RoboDK station: plane_optimization.rdk

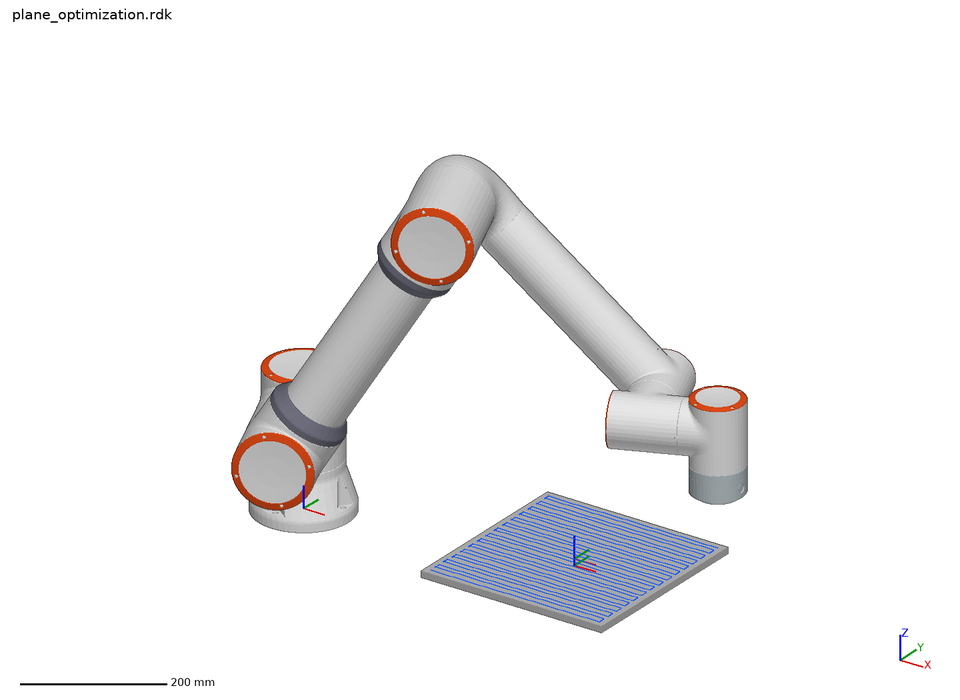
[picture v0: the station drawn from its stored meshes, robots at their saved joint values, targets as dots, program paths as lines]
Station plane_optimization (saved by RoboDK 6.0.4). Poses are relative to the parent item; angles as X-Y-Z fixed-axis rotations.
  - frame FAIRINO FR5 Base at (0, 0, 0) mm
    - robot FAIRINO FR5: 6 axes
        modified DH rows (alpha deg, a mm, theta deg, d mm): 0, 0, 0, 152; 90, 0, 180, 0; 0, 425, 0, 0; 0, 395, 0, 102; -90, 0, 0, 102; 90, 0, 180, 100
        joint limits [-175, -265, -160, -265, -175, -175] to [175, 85, 160, 85, 175, 175]; home [0, -90, -90, 0, 90, 0]; saved at [23.033, -121.455, -104.631, -43.915, 90, 23.033]
      - tool Tool 1, TCP at (0, 0, 80) mm
  - frame PlateFrame at (450, 0, 50) mm
    - target Home (Cartesian target) at (45, -102, 629) mm, rotated rx -90 ry 0 rz -90 deg; joints [0, -90, -90, 0, 90, 0] of FAIRINO FR5
    - target Target_001 (Cartesian target) at (-140, -140, 0) mm, rotated rx -180 ry 0 rz -90 deg; joints [-6.855, -94.267, -146.837, -28.896, 90, -6.855] of FAIRINO FR5
    - target Target_002 (Cartesian target) at (-130, -140, 0) mm, rotated rx -180 ry 0 rz -90 deg; joints [-6.65, -95.39, -145.504, -29.106, 90, -6.65] of FAIRINO FR5
    - target Target_003 (Cartesian target) at (-120, -140, 0) mm, rotated rx -180 ry 0 rz -90 deg; joints [-6.457, -96.486, -144.158, -29.356, 90, -6.457] of FAIRINO FR5
    - target Target_004 (Cartesian target) at (-110, -140, 0) mm, rotated rx -180 ry 0 rz -90 deg; joints [-6.275, -97.559, -142.799, -29.642, 90, -6.275] of FAIRINO FR5
    - target Target_005 (Cartesian target) at (-100, -140, 0) mm, rotated rx -180 ry 0 rz -90 deg; joints [-6.102, -98.61, -141.428, -29.962, 90, -6.102] of FAIRINO FR5
    - target Target_006 (Cartesian target) at (-90, -140, 0) mm, rotated rx -180 ry 0 rz -90 deg; joints [-5.939, -99.642, -140.044, -30.313, 90, -5.939] of FAIRINO FR5
    - target Target_007 (Cartesian target) at (-80, -140, 0) mm, rotated rx -180 ry 0 rz -90 deg; joints [-5.784, -100.658, -138.649, -30.693, 90, -5.784] of FAIRINO FR5
    - target Target_008 (Cartesian target) at (-70, -140, 0) mm, rotated rx -180 ry 0 rz -90 deg; joints [-5.637, -101.66, -137.242, -31.099, 90, -5.637] of FAIRINO FR5
    - target Target_009 (Cartesian target) at (-60, -140, 0) mm, rotated rx -180 ry 0 rz -90 deg; joints [-5.497, -102.648, -135.823, -31.529, 90, -5.497] of FAIRINO FR5
    - target Target_010 (Cartesian target) at (-50, -140, 0) mm, rotated rx -180 ry 0 rz -90 deg; joints [-5.363, -103.625, -134.392, -31.983, 90, -5.363] of FAIRINO FR5
    - target Target_011 (Cartesian target) at (-40, -140, 0) mm, rotated rx -180 ry 0 rz -90 deg; joints [-5.236, -104.592, -132.949, -32.459, 90, -5.236] of FAIRINO FR5
    - target Target_012 (Cartesian target) at (-30, -140, 0) mm, rotated rx -180 ry 0 rz -90 deg; joints [-5.115, -105.55, -131.495, -32.955, 90, -5.115] of FAIRINO FR5
    - target Target_013 (Cartesian target) at (-20, -140, 0) mm, rotated rx -180 ry 0 rz -90 deg; joints [-4.999, -106.501, -130.028, -33.471, 90, -4.999] of FAIRINO FR5
    - target Target_014 (Cartesian target) at (-10, -140, 0) mm, rotated rx -180 ry 0 rz -90 deg; joints [-4.888, -107.446, -128.549, -34.005, 90, -4.888] of FAIRINO FR5
    - target Target_015 (Cartesian target) at (0, -140, 0) mm, rotated rx -180 ry 0 rz -90 deg; joints [-4.782, -108.386, -127.057, -34.557, 90, -4.782] of FAIRINO FR5
    - target Target_016 (Cartesian target) at (10, -140, 0) mm, rotated rx -180 ry 0 rz -90 deg; joints [-4.68, -109.321, -125.553, -35.126, 90, -4.68] of FAIRINO FR5
    - target Target_017 (Cartesian target) at (20, -140, 0) mm, rotated rx -180 ry 0 rz -90 deg; joints [-4.583, -110.253, -124.035, -35.712, 90, -4.583] of FAIRINO FR5
    - target Target_018 (Cartesian target) at (30, -140, 0) mm, rotated rx -180 ry 0 rz -90 deg; joints [-4.489, -111.182, -122.505, -36.314, 90, -4.489] of FAIRINO FR5
    - target Target_019 (Cartesian target) at (40, -140, 0) mm, rotated rx -180 ry 0 rz -90 deg; joints [-4.399, -112.109, -120.96, -36.931, 90, -4.399] of FAIRINO FR5
    - target Target_020 (Cartesian target) at (50, -140, 0) mm, rotated rx -180 ry 0 rz -90 deg; joints [-4.313, -113.036, -119.401, -37.563, 90, -4.313] of FAIRINO FR5
    - target Target_021 (Cartesian target) at (60, -140, 0) mm, rotated rx -180 ry 0 rz -90 deg; joints [-4.23, -113.963, -117.827, -38.21, 90, -4.23] of FAIRINO FR5
    - target Target_022 (Cartesian target) at (70, -140, 0) mm, rotated rx -180 ry 0 rz -90 deg; joints [-4.15, -114.89, -116.238, -38.872, 90, -4.15] of FAIRINO FR5
    - target Target_023 (Cartesian target) at (80, -140, 0) mm, rotated rx -180 ry 0 rz -90 deg; joints [-4.073, -115.818, -114.633, -39.549, 90, -4.073] of FAIRINO FR5
    - target Target_024 (Cartesian target) at (90, -140, 0) mm, rotated rx -180 ry 0 rz -90 deg; joints [-3.999, -116.749, -113.011, -40.24, 90, -3.999] of FAIRINO FR5
    - target Target_025 (Cartesian target) at (100, -140, 0) mm, rotated rx -180 ry 0 rz -90 deg; joints [-3.927, -117.682, -111.373, -40.946, 90, -3.927] of FAIRINO FR5
    - target Target_026 (Cartesian target) at (110, -140, 0) mm, rotated rx -180 ry 0 rz -90 deg; joints [-3.858, -118.618, -109.716, -41.666, 90, -3.858] of FAIRINO FR5
    - target Target_027 (Cartesian target) at (120, -140, 0) mm, rotated rx -180 ry 0 rz -90 deg; joints [-3.792, -119.559, -108.041, -42.401, 90, -3.792] of FAIRINO FR5
    - target Target_028 (Cartesian target) at (130, -140, 0) mm, rotated rx -180 ry 0 rz -90 deg; joints [-3.727, -120.504, -106.346, -43.15, 90, -3.727] of FAIRINO FR5
    - target Target_029 (Cartesian target) at (140, -140, 0) mm, rotated rx -180 ry 0 rz -90 deg; joints [-3.665, -121.455, -104.631, -43.915, 90, -3.665] of FAIRINO FR5
    - target Target_030 (Cartesian target) at (140, -130, 0) mm, rotated rx -180 ry 0 rz -90 deg; joints [-2.706, -121.236, -105.026, -43.738, 90, -2.706] of FAIRINO FR5
    - target Target_031 (Cartesian target) at (130, -130, 0) mm, rotated rx -180 ry 0 rz -90 deg; joints [-2.752, -120.283, -106.743, -42.974, 90, -2.752] of FAIRINO FR5
    - target Target_032 (Cartesian target) at (120, -130, 0) mm, rotated rx -180 ry 0 rz -90 deg; joints [-2.8, -119.335, -108.44, -42.225, 90, -2.8] of FAIRINO FR5
    - target Target_033 (Cartesian target) at (110, -130, 0) mm, rotated rx -180 ry 0 rz -90 deg; joints [-2.85, -118.391, -110.118, -41.491, 90, -2.85] of FAIRINO FR5
    - target Target_034 (Cartesian target) at (100, -130, 0) mm, rotated rx -180 ry 0 rz -90 deg; joints [-2.901, -117.452, -111.777, -40.771, 90, -2.901] of FAIRINO FR5
    - target Target_035 (Cartesian target) at (90, -130, 0) mm, rotated rx -180 ry 0 rz -90 deg; joints [-2.954, -116.515, -113.419, -40.066, 90, -2.954] of FAIRINO FR5
    - target Target_036 (Cartesian target) at (80, -130, 0) mm, rotated rx -180 ry 0 rz -90 deg; joints [-3.009, -115.581, -115.044, -39.375, 90, -3.009] of FAIRINO FR5
    - target Target_037 (Cartesian target) at (70, -130, 0) mm, rotated rx -180 ry 0 rz -90 deg; joints [-3.066, -114.648, -116.653, -38.699, 90, -3.066] of FAIRINO FR5
    - target Target_038 (Cartesian target) at (60, -130, 0) mm, rotated rx -180 ry 0 rz -90 deg; joints [-3.125, -113.717, -118.246, -38.037, 90, -3.125] of FAIRINO FR5
    - target Target_039 (Cartesian target) at (50, -130, 0) mm, rotated rx -180 ry 0 rz -90 deg; joints [-3.187, -112.785, -119.824, -37.39, 90, -3.187] of FAIRINO FR5
    - target Target_040 (Cartesian target) at (40, -130, 0) mm, rotated rx -180 ry 0 rz -90 deg; joints [-3.251, -111.853, -121.388, -36.759, 90, -3.251] of FAIRINO FR5
    - target Target_041 (Cartesian target) at (30, -130, 0) mm, rotated rx -180 ry 0 rz -90 deg; joints [-3.318, -110.92, -122.938, -36.142, 90, -3.318] of FAIRINO FR5
    - target Target_042 (Cartesian target) at (20, -130, 0) mm, rotated rx -180 ry 0 rz -90 deg; joints [-3.388, -109.984, -124.474, -35.542, 90, -3.388] of FAIRINO FR5
    - target Target_043 (Cartesian target) at (10, -130, 0) mm, rotated rx -180 ry 0 rz -90 deg; joints [-3.46, -109.046, -125.997, -34.957, 90, -3.46] of FAIRINO FR5
    - target Target_044 (Cartesian target) at (0, -130, 0) mm, rotated rx -180 ry 0 rz -90 deg; joints [-3.536, -108.103, -127.508, -34.389, 90, -3.536] of FAIRINO FR5
    - target Target_045 (Cartesian target) at (-10, -130, 0) mm, rotated rx -180 ry 0 rz -90 deg; joints [-3.615, -107.156, -129.006, -33.839, 90, -3.615] of FAIRINO FR5
    - target Target_046 (Cartesian target) at (-20, -130, 0) mm, rotated rx -180 ry 0 rz -90 deg; joints [-3.697, -106.202, -130.491, -33.306, 90, -3.697] of FAIRINO FR5
    - target Target_047 (Cartesian target) at (-30, -130, 0) mm, rotated rx -180 ry 0 rz -90 deg; joints [-3.784, -105.242, -131.965, -32.793, 90, -3.784] of FAIRINO FR5
    - target Target_048 (Cartesian target) at (-40, -130, 0) mm, rotated rx -180 ry 0 rz -90 deg; joints [-3.874, -104.273, -133.428, -32.299, 90, -3.874] of FAIRINO FR5
    - target Target_049 (Cartesian target) at (-50, -130, 0) mm, rotated rx -180 ry 0 rz -90 deg; joints [-3.969, -103.295, -134.878, -31.827, 90, -3.969] of FAIRINO FR5
    - target Target_050 (Cartesian target) at (-60, -130, 0) mm, rotated rx -180 ry 0 rz -90 deg; joints [-4.069, -102.306, -136.318, -31.377, 90, -4.069] of FAIRINO FR5
    - target Target_051 (Cartesian target) at (-70, -130, 0) mm, rotated rx -180 ry 0 rz -90 deg; joints [-4.174, -101.304, -137.745, -30.951, 90, -4.174] of FAIRINO FR5
    - target Target_052 (Cartesian target) at (-80, -130, 0) mm, rotated rx -180 ry 0 rz -90 deg; joints [-4.284, -100.288, -139.162, -30.55, 90, -4.284] of FAIRINO FR5
    - target Target_053 (Cartesian target) at (-90, -130, 0) mm, rotated rx -180 ry 0 rz -90 deg; joints [-4.4, -99.255, -140.567, -30.177, 90, -4.4] of FAIRINO FR5
    - target Target_054 (Cartesian target) at (-100, -130, 0) mm, rotated rx -180 ry 0 rz -90 deg; joints [-4.522, -98.205, -141.961, -29.834, 90, -4.522] of FAIRINO FR5
    - target Target_055 (Cartesian target) at (-110, -130, 0) mm, rotated rx -180 ry 0 rz -90 deg; joints [-4.651, -97.133, -143.343, -29.524, 90, -4.651] of FAIRINO FR5
    - target Target_056 (Cartesian target) at (-120, -130, 0) mm, rotated rx -180 ry 0 rz -90 deg; joints [-4.788, -96.038, -144.714, -29.248, 90, -4.788] of FAIRINO FR5
    - target Target_057 (Cartesian target) at (-130, -130, 0) mm, rotated rx -180 ry 0 rz -90 deg; joints [-4.933, -94.917, -146.072, -29.012, 90, -4.933] of FAIRINO FR5
    - target Target_058 (Cartesian target) at (-140, -130, 0) mm, rotated rx -180 ry 0 rz -90 deg; joints [-5.087, -93.765, -147.417, -28.818, 90, -5.087] of FAIRINO FR5
    - target Target_059 (Cartesian target) at (-140, -120, 0) mm, rotated rx -180 ry 0 rz -90 deg; joints [-3.292, -93.288, -147.96, -28.752, 90, -3.292] of FAIRINO FR5
    - target Target_060 (Cartesian target) at (-130, -120, 0) mm, rotated rx -180 ry 0 rz -90 deg; joints [-3.191, -94.468, -146.602, -28.93, 90, -3.191] of FAIRINO FR5
    - target Target_061 (Cartesian target) at (-120, -120, 0) mm, rotated rx -180 ry 0 rz -90 deg; joints [-3.096, -95.614, -145.233, -29.153, 90, -3.096] of FAIRINO FR5
    - target Target_062 (Cartesian target) at (-110, -120, 0) mm, rotated rx -180 ry 0 rz -90 deg; joints [-3.007, -96.731, -143.851, -29.417, 90, -3.007] of FAIRINO FR5
    - target Target_063 (Cartesian target) at (-100, -120, 0) mm, rotated rx -180 ry 0 rz -90 deg; joints [-2.922, -97.822, -142.459, -29.719, 90, -2.922] of FAIRINO FR5
    - target Target_064 (Cartesian target) at (-90, -120, 0) mm, rotated rx -180 ry 0 rz -90 deg; joints [-2.842, -98.891, -141.055, -30.054, 90, -2.842] of FAIRINO FR5
    - target Target_065 (Cartesian target) at (-80, -120, 0) mm, rotated rx -180 ry 0 rz -90 deg; joints [-2.767, -99.939, -139.64, -30.42, 90, -2.767] of FAIRINO FR5
    - target Target_066 (Cartesian target) at (-70, -120, 0) mm, rotated rx -180 ry 0 rz -90 deg; joints [-2.695, -100.97, -138.215, -30.816, 90, -2.695] of FAIRINO FR5
    - target Target_067 (Cartesian target) at (-60, -120, 0) mm, rotated rx -180 ry 0 rz -90 deg; joints [-2.627, -101.985, -136.778, -31.237, 90, -2.627] of FAIRINO FR5
    - target Target_068 (Cartesian target) at (-50, -120, 0) mm, rotated rx -180 ry 0 rz -90 deg; joints [-2.562, -102.986, -135.331, -31.683, 90, -2.562] of FAIRINO FR5
    - target Target_069 (Cartesian target) at (-40, -120, 0) mm, rotated rx -180 ry 0 rz -90 deg; joints [-2.5, -103.975, -133.873, -32.152, 90, -2.5] of FAIRINO FR5
    - target Target_070 (Cartesian target) at (-30, -120, 0) mm, rotated rx -180 ry 0 rz -90 deg; joints [-2.441, -104.953, -132.403, -32.643, 90, -2.441] of FAIRINO FR5
    - target Target_071 (Cartesian target) at (-20, -120, 0) mm, rotated rx -180 ry 0 rz -90 deg; joints [-2.385, -105.923, -130.922, -33.155, 90, -2.385] of FAIRINO FR5
    - target Target_072 (Cartesian target) at (-10, -120, 0) mm, rotated rx -180 ry 0 rz -90 deg; joints [-2.332, -106.885, -129.43, -33.685, 90, -2.332] of FAIRINO FR5
    - target Target_073 (Cartesian target) at (0, -120, 0) mm, rotated rx -180 ry 0 rz -90 deg; joints [-2.28, -107.84, -127.926, -34.234, 90, -2.28] of FAIRINO FR5
    - target Target_074 (Cartesian target) at (10, -120, 0) mm, rotated rx -180 ry 0 rz -90 deg; joints [-2.231, -108.789, -126.41, -34.801, 90, -2.231] of FAIRINO FR5
    - target Target_075 (Cartesian target) at (20, -120, 0) mm, rotated rx -180 ry 0 rz -90 deg; joints [-2.184, -109.734, -124.882, -35.384, 90, -2.184] of FAIRINO FR5
    - target Target_076 (Cartesian target) at (30, -120, 0) mm, rotated rx -180 ry 0 rz -90 deg; joints [-2.139, -110.676, -123.34, -35.984, 90, -2.139] of FAIRINO FR5
    - target Target_077 (Cartesian target) at (40, -120, 0) mm, rotated rx -180 ry 0 rz -90 deg; joints [-2.096, -111.615, -121.786, -36.6, 90, -2.096] of FAIRINO FR5
    - target Target_078 (Cartesian target) at (50, -120, 0) mm, rotated rx -180 ry 0 rz -90 deg; joints [-2.054, -112.552, -120.218, -37.231, 90, -2.054] of FAIRINO FR5
    - target Target_079 (Cartesian target) at (60, -120, 0) mm, rotated rx -180 ry 0 rz -90 deg; joints [-2.014, -113.488, -118.635, -37.877, 90, -2.014] of FAIRINO FR5
    - target Target_080 (Cartesian target) at (70, -120, 0) mm, rotated rx -180 ry 0 rz -90 deg; joints [-1.976, -114.424, -117.038, -38.538, 90, -1.976] of FAIRINO FR5
    - target Target_081 (Cartesian target) at (80, -120, 0) mm, rotated rx -180 ry 0 rz -90 deg; joints [-1.939, -115.36, -115.426, -39.214, 90, -1.939] of FAIRINO FR5
    - target Target_082 (Cartesian target) at (90, -120, 0) mm, rotated rx -180 ry 0 rz -90 deg; joints [-1.903, -116.298, -113.798, -39.904, 90, -1.903] of FAIRINO FR5
    - target Target_083 (Cartesian target) at (100, -120, 0) mm, rotated rx -180 ry 0 rz -90 deg; joints [-1.869, -117.238, -112.153, -40.609, 90, -1.869] of FAIRINO FR5
    - target Target_084 (Cartesian target) at (110, -120, 0) mm, rotated rx -180 ry 0 rz -90 deg; joints [-1.836, -118.181, -110.491, -41.328, 90, -1.836] of FAIRINO FR5
    - target Target_085 (Cartesian target) at (120, -120, 0) mm, rotated rx -180 ry 0 rz -90 deg; joints [-1.804, -119.127, -108.81, -42.062, 90, -1.804] of FAIRINO FR5
    - target Target_086 (Cartesian target) at (130, -120, 0) mm, rotated rx -180 ry 0 rz -90 deg; joints [-1.773, -120.078, -107.111, -42.811, 90, -1.773] of FAIRINO FR5
    - target Target_087 (Cartesian target) at (140, -120, 0) mm, rotated rx -180 ry 0 rz -90 deg; joints [-1.743, -121.033, -105.392, -43.575, 90, -1.743] of FAIRINO FR5
    - target Target_088 (Cartesian target) at (140, -110, 0) mm, rotated rx -180 ry 0 rz -90 deg; joints [-0.776, -120.846, -105.729, -43.424, 90, -0.776] of FAIRINO FR5
    - target Target_089 (Cartesian target) at (130, -110, 0) mm, rotated rx -180 ry 0 rz -90 deg; joints [-0.789, -119.889, -107.45, -42.661, 90, -0.789] of FAIRINO FR5
    - target Target_090 (Cartesian target) at (120, -110, 0) mm, rotated rx -180 ry 0 rz -90 deg; joints [-0.803, -118.936, -109.152, -41.913, 90, -0.803] of FAIRINO FR5
    - target Target_091 (Cartesian target) at (110, -110, 0) mm, rotated rx -180 ry 0 rz -90 deg; joints [-0.817, -117.987, -110.834, -41.179, 90, -0.817] of FAIRINO FR5
    - target Target_092 (Cartesian target) at (100, -110, 0) mm, rotated rx -180 ry 0 rz -90 deg; joints [-0.832, -117.041, -112.499, -40.46, 90, -0.832] of FAIRINO FR5
    - target Target_093 (Cartesian target) at (90, -110, 0) mm, rotated rx -180 ry 0 rz -90 deg; joints [-0.848, -116.098, -114.147, -39.755, 90, -0.848] of FAIRINO FR5
    - target Target_094 (Cartesian target) at (80, -110, 0) mm, rotated rx -180 ry 0 rz -90 deg; joints [-0.864, -115.157, -115.778, -39.066, 90, -0.864] of FAIRINO FR5
    - target Target_095 (Cartesian target) at (70, -110, 0) mm, rotated rx -180 ry 0 rz -90 deg; joints [-0.88, -114.216, -117.393, -38.39, 90, -0.88] of FAIRINO FR5
    - target Target_096 (Cartesian target) at (60, -110, 0) mm, rotated rx -180 ry 0 rz -90 deg; joints [-0.897, -113.276, -118.994, -37.729, 90, -0.897] of FAIRINO FR5
    - target Target_097 (Cartesian target) at (50, -110, 0) mm, rotated rx -180 ry 0 rz -90 deg; joints [-0.915, -112.336, -120.58, -37.084, 90, -0.915] of FAIRINO FR5
    - target Target_098 (Cartesian target) at (40, -110, 0) mm, rotated rx -180 ry 0 rz -90 deg; joints [-0.934, -111.394, -122.153, -36.453, 90, -0.934] of FAIRINO FR5
    - target Target_099 (Cartesian target) at (30, -110, 0) mm, rotated rx -180 ry 0 rz -90 deg; joints [-0.953, -110.45, -123.712, -35.838, 90, -0.953] of FAIRINO FR5
    - target Target_100 (Cartesian target) at (20, -110, 0) mm, rotated rx -180 ry 0 rz -90 deg; joints [-0.973, -109.503, -125.258, -35.239, 90, -0.973] of FAIRINO FR5
    - target Target_101 (Cartesian target) at (10, -110, 0) mm, rotated rx -180 ry 0 rz -90 deg; joints [-0.994, -108.552, -126.791, -34.657, 90, -0.994] of FAIRINO FR5
    - target Target_102 (Cartesian target) at (0, -110, 0) mm, rotated rx -180 ry 0 rz -90 deg; joints [-1.016, -107.596, -128.313, -34.092, 90, -1.016] of FAIRINO FR5
    - target Target_103 (Cartesian target) at (-10, -110, 0) mm, rotated rx -180 ry 0 rz -90 deg; joints [-1.039, -106.633, -129.823, -33.544, 90, -1.039] of FAIRINO FR5
    - target Target_104 (Cartesian target) at (-20, -110, 0) mm, rotated rx -180 ry 0 rz -90 deg; joints [-1.064, -105.664, -131.321, -33.015, 90, -1.064] of FAIRINO FR5
    - target Target_105 (Cartesian target) at (-30, -110, 0) mm, rotated rx -180 ry 0 rz -90 deg; joints [-1.089, -104.686, -132.808, -32.506, 90, -1.089] of FAIRINO FR5
    - target Target_106 (Cartesian target) at (-40, -110, 0) mm, rotated rx -180 ry 0 rz -90 deg; joints [-1.115, -103.698, -134.284, -32.018, 90, -1.115] of FAIRINO FR5
    - target Target_107 (Cartesian target) at (-50, -110, 0) mm, rotated rx -180 ry 0 rz -90 deg; joints [-1.143, -102.698, -135.75, -31.552, 90, -1.143] of FAIRINO FR5
    - target Target_108 (Cartesian target) at (-60, -110, 0) mm, rotated rx -180 ry 0 rz -90 deg; joints [-1.172, -101.686, -137.205, -31.11, 90, -1.172] of FAIRINO FR5
    - target Target_109 (Cartesian target) at (-70, -110, 0) mm, rotated rx -180 ry 0 rz -90 deg; joints [-1.203, -100.658, -138.649, -30.693, 90, -1.203] of FAIRINO FR5
    - target Target_110 (Cartesian target) at (-80, -110, 0) mm, rotated rx -180 ry 0 rz -90 deg; joints [-1.235, -99.614, -140.083, -30.303, 90, -1.235] of FAIRINO FR5
    - target Target_111 (Cartesian target) at (-90, -110, 0) mm, rotated rx -180 ry 0 rz -90 deg; joints [-1.269, -98.55, -141.507, -29.943, 90, -1.269] of FAIRINO FR5
    - target Target_112 (Cartesian target) at (-100, -110, 0) mm, rotated rx -180 ry 0 rz -90 deg; joints [-1.305, -97.465, -142.92, -29.615, 90, -1.305] of FAIRINO FR5
    - target Target_113 (Cartesian target) at (-110, -110, 0) mm, rotated rx -180 ry 0 rz -90 deg; joints [-1.343, -96.355, -144.322, -29.323, 90, -1.343] of FAIRINO FR5
    - target Target_114 (Cartesian target) at (-120, -110, 0) mm, rotated rx -180 ry 0 rz -90 deg; joints [-1.384, -95.216, -145.714, -29.07, 90, -1.384] of FAIRINO FR5
    - target Target_115 (Cartesian target) at (-130, -110, 0) mm, rotated rx -180 ry 0 rz -90 deg; joints [-1.426, -94.045, -147.094, -28.86, 90, -1.426] of FAIRINO FR5
    - target Target_116 (Cartesian target) at (-140, -110, 0) mm, rotated rx -180 ry 0 rz -90 deg; joints [-1.472, -92.838, -148.463, -28.698, 90, -1.472] of FAIRINO FR5
    - target Target_117 (Cartesian target) at (-140, -100, 0) mm, rotated rx -180 ry 0 rz -90 deg; joints [0.37, -92.418, -148.927, -28.655, 90, 0.37] of FAIRINO FR5
    - target Target_118 (Cartesian target) at (-130, -100, 0) mm, rotated rx -180 ry 0 rz -90 deg; joints [0.358, -93.652, -147.547, -28.801, 90, 0.358] of FAIRINO FR5
    - target Target_119 (Cartesian target) at (-120, -100, 0) mm, rotated rx -180 ry 0 rz -90 deg; joints [0.348, -94.845, -146.156, -28.998, 90, 0.348] of FAIRINO FR5
    - target Target_120 (Cartesian target) at (-110, -100, 0) mm, rotated rx -180 ry 0 rz -90 deg; joints [0.337, -96.005, -144.755, -29.24, 90, 0.337] of FAIRINO FR5
    - target Target_121 (Cartesian target) at (-100, -100, 0) mm, rotated rx -180 ry 0 rz -90 deg; joints [0.328, -97.133, -143.343, -29.524, 90, 0.328] of FAIRINO FR5
    - target Target_122 (Cartesian target) at (-90, -100, 0) mm, rotated rx -180 ry 0 rz -90 deg; joints [0.319, -98.235, -141.922, -29.844, 90, 0.319] of FAIRINO FR5
    - target Target_123 (Cartesian target) at (-80, -100, 0) mm, rotated rx -180 ry 0 rz -90 deg; joints [0.31, -99.313, -140.49, -30.197, 90, 0.31] of FAIRINO FR5
    - target Target_124 (Cartesian target) at (-70, -100, 0) mm, rotated rx -180 ry 0 rz -90 deg; joints [0.302, -100.37, -139.048, -30.582, 90, 0.302] of FAIRINO FR5
    - target Target_125 (Cartesian target) at (-60, -100, 0) mm, rotated rx -180 ry 0 rz -90 deg; joints [0.294, -101.41, -137.596, -30.994, 90, 0.294] of FAIRINO FR5
    - target Target_126 (Cartesian target) at (-50, -100, 0) mm, rotated rx -180 ry 0 rz -90 deg; joints [0.287, -102.433, -136.134, -31.433, 90, 0.287] of FAIRINO FR5
    - target Target_127 (Cartesian target) at (-40, -100, 0) mm, rotated rx -180 ry 0 rz -90 deg; joints [0.28, -103.442, -134.662, -31.896, 90, 0.28] of FAIRINO FR5
    - target Target_128 (Cartesian target) at (-30, -100, 0) mm, rotated rx -180 ry 0 rz -90 deg; joints [0.273, -104.439, -133.179, -32.382, 90, 0.273] of FAIRINO FR5
    - target Target_129 (Cartesian target) at (-20, -100, 0) mm, rotated rx -180 ry 0 rz -90 deg; joints [0.267, -105.425, -131.686, -32.889, 90, 0.267] of FAIRINO FR5
    - target Target_130 (Cartesian target) at (-10, -100, 0) mm, rotated rx -180 ry 0 rz -90 deg; joints [0.261, -106.402, -130.182, -33.416, 90, 0.261] of FAIRINO FR5
    - target Target_131 (Cartesian target) at (0, -100, 0) mm, rotated rx -180 ry 0 rz -90 deg; joints [0.255, -107.371, -128.667, -33.962, 90, 0.255] of FAIRINO FR5
    - target Target_132 (Cartesian target) at (10, -100, 0) mm, rotated rx -180 ry 0 rz -90 deg; joints [0.249, -108.333, -127.141, -34.526, 90, 0.249] of FAIRINO FR5
    - target Target_133 (Cartesian target) at (20, -100, 0) mm, rotated rx -180 ry 0 rz -90 deg; joints [0.244, -109.29, -125.602, -35.108, 90, 0.244] of FAIRINO FR5
    - target Target_134 (Cartesian target) at (30, -100, 0) mm, rotated rx -180 ry 0 rz -90 deg; joints [0.239, -110.243, -124.052, -35.706, 90, 0.239] of FAIRINO FR5
    - target Target_135 (Cartesian target) at (40, -100, 0) mm, rotated rx -180 ry 0 rz -90 deg; joints [0.234, -111.192, -122.489, -36.32, 90, 0.234] of FAIRINO FR5
    - target Target_136 (Cartesian target) at (50, -100, 0) mm, rotated rx -180 ry 0 rz -90 deg; joints [0.229, -112.138, -120.912, -36.95, 90, 0.229] of FAIRINO FR5
    - target Target_137 (Cartesian target) at (60, -100, 0) mm, rotated rx -180 ry 0 rz -90 deg; joints [0.225, -113.082, -119.323, -37.595, 90, 0.225] of FAIRINO FR5
    - target Target_138 (Cartesian target) at (70, -100, 0) mm, rotated rx -180 ry 0 rz -90 deg; joints [0.22, -114.026, -117.719, -38.255, 90, 0.22] of FAIRINO FR5
    - target Target_139 (Cartesian target) at (80, -100, 0) mm, rotated rx -180 ry 0 rz -90 deg; joints [0.216, -114.97, -116.1, -38.93, 90, 0.216] of FAIRINO FR5
    - target Target_140 (Cartesian target) at (90, -100, 0) mm, rotated rx -180 ry 0 rz -90 deg; joints [0.212, -115.914, -114.466, -39.62, 90, 0.212] of FAIRINO FR5
    - target Target_141 (Cartesian target) at (100, -100, 0) mm, rotated rx -180 ry 0 rz -90 deg; joints [0.208, -116.861, -112.815, -40.324, 90, 0.208] of FAIRINO FR5
    - target Target_142 (Cartesian target) at (110, -100, 0) mm, rotated rx -180 ry 0 rz -90 deg; joints [0.205, -117.809, -111.148, -41.043, 90, 0.205] of FAIRINO FR5
    - target Target_143 (Cartesian target) at (120, -100, 0) mm, rotated rx -180 ry 0 rz -90 deg; joints [0.201, -118.76, -109.463, -41.776, 90, 0.201] of FAIRINO FR5
    - target Target_144 (Cartesian target) at (130, -100, 0) mm, rotated rx -180 ry 0 rz -90 deg; joints [0.198, -119.716, -107.76, -42.524, 90, 0.198] of FAIRINO FR5
    - target Target_145 (Cartesian target) at (140, -100, 0) mm, rotated rx -180 ry 0 rz -90 deg; joints [0.194, -120.675, -106.037, -43.287, 90, 0.194] of FAIRINO FR5
    - target Target_146 (Cartesian target) at (140, -90, 0) mm, rotated rx -180 ry 0 rz -90 deg; joints [1.167, -120.52, -106.317, -43.163, 90, 1.167] of FAIRINO FR5
    - target Target_147 (Cartesian target) at (130, -90, 0) mm, rotated rx -180 ry 0 rz -90 deg; joints [1.187, -119.559, -108.041, -42.401, 90, 1.187] of FAIRINO FR5
    - target Target_148 (Cartesian target) at (120, -90, 0) mm, rotated rx -180 ry 0 rz -90 deg; joints [1.208, -118.601, -109.746, -41.653, 90, 1.208] of FAIRINO FR5
    - target Target_149 (Cartesian target) at (110, -90, 0) mm, rotated rx -180 ry 0 rz -90 deg; joints [1.23, -117.648, -111.433, -40.92, 90, 1.23] of FAIRINO FR5
    - target Target_150 (Cartesian target) at (100, -90, 0) mm, rotated rx -180 ry 0 rz -90 deg; joints [1.252, -116.697, -113.102, -40.201, 90, 1.252] of FAIRINO FR5
    - target Target_151 (Cartesian target) at (90, -90, 0) mm, rotated rx -180 ry 0 rz -90 deg; joints [1.276, -115.748, -114.755, -39.497, 90, 1.276] of FAIRINO FR5
    - target Target_152 (Cartesian target) at (80, -90, 0) mm, rotated rx -180 ry 0 rz -90 deg; joints [1.3, -114.8, -116.392, -38.808, 90, 1.3] of FAIRINO FR5
    - target Target_153 (Cartesian target) at (70, -90, 0) mm, rotated rx -180 ry 0 rz -90 deg; joints [1.325, -113.854, -118.013, -38.133, 90, 1.325] of FAIRINO FR5
    - target Target_154 (Cartesian target) at (60, -90, 0) mm, rotated rx -180 ry 0 rz -90 deg; joints [1.351, -112.906, -119.62, -37.473, 90, 1.351] of FAIRINO FR5
    - target Target_155 (Cartesian target) at (50, -90, 0) mm, rotated rx -180 ry 0 rz -90 deg; joints [1.378, -111.958, -121.213, -36.829, 90, 1.378] of FAIRINO FR5
    - target Target_156 (Cartesian target) at (40, -90, 0) mm, rotated rx -180 ry 0 rz -90 deg; joints [1.406, -111.007, -122.793, -36.199, 90, 1.406] of FAIRINO FR5
    - target Target_157 (Cartesian target) at (30, -90, 0) mm, rotated rx -180 ry 0 rz -90 deg; joints [1.436, -110.054, -124.36, -35.586, 90, 1.436] of FAIRINO FR5
    - target Target_158 (Cartesian target) at (20, -90, 0) mm, rotated rx -180 ry 0 rz -90 deg; joints [1.467, -109.097, -125.915, -34.988, 90, 1.467] of FAIRINO FR5
    - target Target_159 (Cartesian target) at (10, -90, 0) mm, rotated rx -180 ry 0 rz -90 deg; joints [1.499, -108.135, -127.457, -34.408, 90, 1.499] of FAIRINO FR5
    - target Target_160 (Cartesian target) at (0, -90, 0) mm, rotated rx -180 ry 0 rz -90 deg; joints [1.532, -107.167, -128.989, -33.845, 90, 1.532] of FAIRINO FR5
    - target Target_161 (Cartesian target) at (-10, -90, 0) mm, rotated rx -180 ry 0 rz -90 deg; joints [1.567, -106.191, -130.509, -33.3, 90, 1.567] of FAIRINO FR5
    - target Target_162 (Cartesian target) at (-20, -90, 0) mm, rotated rx -180 ry 0 rz -90 deg; joints [1.604, -105.207, -132.018, -32.775, 90, 1.604] of FAIRINO FR5
    - target Target_163 (Cartesian target) at (-30, -90, 0) mm, rotated rx -180 ry 0 rz -90 deg; joints [1.642, -104.214, -133.516, -32.27, 90, 1.642] of FAIRINO FR5
    - target Target_164 (Cartesian target) at (-40, -90, 0) mm, rotated rx -180 ry 0 rz -90 deg; joints [1.683, -103.209, -135.005, -31.787, 90, 1.683] of FAIRINO FR5
    - target Target_165 (Cartesian target) at (-50, -90, 0) mm, rotated rx -180 ry 0 rz -90 deg; joints [1.725, -102.19, -136.483, -31.326, 90, 1.725] of FAIRINO FR5
    - target Target_166 (Cartesian target) at (-60, -90, 0) mm, rotated rx -180 ry 0 rz -90 deg; joints [1.77, -101.157, -137.952, -30.891, 90, 1.77] of FAIRINO FR5
    - target Target_167 (Cartesian target) at (-70, -90, 0) mm, rotated rx -180 ry 0 rz -90 deg; joints [1.816, -100.107, -139.41, -30.483, 90, 1.816] of FAIRINO FR5
    - target Target_168 (Cartesian target) at (-80, -90, 0) mm, rotated rx -180 ry 0 rz -90 deg; joints [1.866, -99.037, -140.86, -30.103, 90, 1.866] of FAIRINO FR5
    - target Target_169 (Cartesian target) at (-90, -90, 0) mm, rotated rx -180 ry 0 rz -90 deg; joints [1.918, -97.945, -142.299, -29.755, 90, 1.918] of FAIRINO FR5
    - target Target_170 (Cartesian target) at (-100, -90, 0) mm, rotated rx -180 ry 0 rz -90 deg; joints [1.974, -96.828, -143.729, -29.443, 90, 1.974] of FAIRINO FR5
    - target Target_171 (Cartesian target) at (-110, -90, 0) mm, rotated rx -180 ry 0 rz -90 deg; joints [2.032, -95.683, -145.149, -29.168, 90, 2.032] of FAIRINO FR5
    - target Target_172 (Cartesian target) at (-120, -90, 0) mm, rotated rx -180 ry 0 rz -90 deg; joints [2.094, -94.504, -146.56, -28.936, 90, 2.094] of FAIRINO FR5
    - target Target_173 (Cartesian target) at (-130, -90, 0) mm, rotated rx -180 ry 0 rz -90 deg; joints [2.161, -93.288, -147.96, -28.752, 90, 2.161] of FAIRINO FR5
    - target Target_174 (Cartesian target) at (-140, -90, 0) mm, rotated rx -180 ry 0 rz -90 deg; joints [2.231, -92.029, -149.349, -28.621, 90, 2.231] of FAIRINO FR5
    - target Target_175 (Cartesian target) at (-140, -80, 0) mm, rotated rx -180 ry 0 rz -90 deg; joints [4.108, -91.674, -149.73, -28.595, 90, 4.108] of FAIRINO FR5
    - target Target_176 (Cartesian target) at (-130, -80, 0) mm, rotated rx -180 ry 0 rz -90 deg; joints [3.977, -92.957, -148.332, -28.712, 90, 3.977] of FAIRINO FR5
    - target Target_177 (Cartesian target) at (-120, -80, 0) mm, rotated rx -180 ry 0 rz -90 deg; joints [3.854, -94.193, -146.923, -28.884, 90, 3.854] of FAIRINO FR5
    - target Target_178 (Cartesian target) at (-110, -80, 0) mm, rotated rx -180 ry 0 rz -90 deg; joints [3.739, -95.39, -145.504, -29.106, 90, 3.739] of FAIRINO FR5
    - target Target_179 (Cartesian target) at (-100, -80, 0) mm, rotated rx -180 ry 0 rz -90 deg; joints [3.63, -96.552, -144.076, -29.372, 90, 3.63] of FAIRINO FR5
    - target Target_180 (Cartesian target) at (-90, -80, 0) mm, rotated rx -180 ry 0 rz -90 deg; joints [3.528, -97.683, -142.639, -29.678, 90, 3.528] of FAIRINO FR5
    - target Target_181 (Cartesian target) at (-80, -80, 0) mm, rotated rx -180 ry 0 rz -90 deg; joints [3.431, -98.788, -141.192, -30.02, 90, 3.431] of FAIRINO FR5
    - target Target_182 (Cartesian target) at (-70, -80, 0) mm, rotated rx -180 ry 0 rz -90 deg; joints [3.339, -99.869, -139.736, -30.395, 90, 3.339] of FAIRINO FR5
    - target Target_183 (Cartesian target) at (-60, -80, 0) mm, rotated rx -180 ry 0 rz -90 deg; joints [3.253, -100.929, -138.271, -30.799, 90, 3.253] of FAIRINO FR5
    - target Target_184 (Cartesian target) at (-50, -80, 0) mm, rotated rx -180 ry 0 rz -90 deg; joints [3.17, -101.972, -136.797, -31.231, 90, 3.17] of FAIRINO FR5
    - target Target_185 (Cartesian target) at (-40, -80, 0) mm, rotated rx -180 ry 0 rz -90 deg; joints [3.092, -102.998, -135.313, -31.689, 90, 3.092] of FAIRINO FR5
    - target Target_186 (Cartesian target) at (-30, -80, 0) mm, rotated rx -180 ry 0 rz -90 deg; joints [3.018, -104.011, -133.819, -32.17, 90, 3.018] of FAIRINO FR5
    - target Target_187 (Cartesian target) at (-20, -80, 0) mm, rotated rx -180 ry 0 rz -90 deg; joints [2.947, -105.011, -132.315, -32.673, 90, 2.947] of FAIRINO FR5
    - target Target_188 (Cartesian target) at (-10, -80, 0) mm, rotated rx -180 ry 0 rz -90 deg; joints [2.879, -106.001, -130.802, -33.197, 90, 2.879] of FAIRINO FR5
    - target Target_189 (Cartesian target) at (0, -80, 0) mm, rotated rx -180 ry 0 rz -90 deg; joints [2.815, -106.983, -129.277, -33.74, 90, 2.815] of FAIRINO FR5
    - target Target_190 (Cartesian target) at (10, -80, 0) mm, rotated rx -180 ry 0 rz -90 deg; joints [2.753, -107.956, -127.742, -34.302, 90, 2.753] of FAIRINO FR5
    - target Target_191 (Cartesian target) at (20, -80, 0) mm, rotated rx -180 ry 0 rz -90 deg; joints [2.694, -108.923, -126.195, -34.882, 90, 2.694] of FAIRINO FR5
    - target Target_192 (Cartesian target) at (30, -80, 0) mm, rotated rx -180 ry 0 rz -90 deg; joints [2.637, -109.885, -124.637, -35.479, 90, 2.637] of FAIRINO FR5
    - target Target_193 (Cartesian target) at (40, -80, 0) mm, rotated rx -180 ry 0 rz -90 deg; joints [2.583, -110.842, -123.066, -36.092, 90, 2.583] of FAIRINO FR5
    - target Target_194 (Cartesian target) at (50, -80, 0) mm, rotated rx -180 ry 0 rz -90 deg; joints [2.531, -111.796, -121.483, -36.72, 90, 2.531] of FAIRINO FR5
    - target Target_195 (Cartesian target) at (60, -80, 0) mm, rotated rx -180 ry 0 rz -90 deg; joints [2.481, -112.748, -119.887, -37.365, 90, 2.481] of FAIRINO FR5
    - target Target_196 (Cartesian target) at (70, -80, 0) mm, rotated rx -180 ry 0 rz -90 deg; joints [2.433, -113.698, -118.277, -38.024, 90, 2.433] of FAIRINO FR5
    - target Target_197 (Cartesian target) at (80, -80, 0) mm, rotated rx -180 ry 0 rz -90 deg; joints [2.387, -114.648, -116.653, -38.699, 90, 2.387] of FAIRINO FR5
    - target Target_198 (Cartesian target) at (90, -80, 0) mm, rotated rx -180 ry 0 rz -90 deg; joints [2.342, -115.599, -115.014, -39.388, 90, 2.342] of FAIRINO FR5
    - target Target_199 (Cartesian target) at (100, -80, 0) mm, rotated rx -180 ry 0 rz -90 deg; joints [2.299, -116.55, -113.359, -40.091, 90, 2.299] of FAIRINO FR5
    - target Target_200 (Cartesian target) at (110, -80, 0) mm, rotated rx -180 ry 0 rz -90 deg; joints [2.258, -117.503, -111.687, -40.81, 90, 2.258] of FAIRINO FR5
    - target Target_201 (Cartesian target) at (120, -80, 0) mm, rotated rx -180 ry 0 rz -90 deg; joints [2.218, -118.459, -109.999, -41.542, 90, 2.218] of FAIRINO FR5
    - target Target_202 (Cartesian target) at (130, -80, 0) mm, rotated rx -180 ry 0 rz -90 deg; joints [2.18, -119.418, -108.292, -42.29, 90, 2.18] of FAIRINO FR5
    - target Target_203 (Cartesian target) at (140, -80, 0) mm, rotated rx -180 ry 0 rz -90 deg; joints [2.142, -120.381, -106.567, -43.052, 90, 2.142] of FAIRINO FR5
    - target Target_204 (Cartesian target) at (140, -70, 0) mm, rotated rx -180 ry 0 rz -90 deg; joints [3.119, -120.258, -106.787, -42.954, 90, 3.119] of FAIRINO FR5
    - target Target_205 (Cartesian target) at (130, -70, 0) mm, rotated rx -180 ry 0 rz -90 deg; joints [3.173, -119.293, -108.514, -42.192, 90, 3.173] of FAIRINO FR5
    - target Target_206 (Cartesian target) at (120, -70, 0) mm, rotated rx -180 ry 0 rz -90 deg; joints [3.229, -118.333, -110.222, -41.445, 90, 3.229] of FAIRINO FR5
    - target Target_207 (Cartesian target) at (110, -70, 0) mm, rotated rx -180 ry 0 rz -90 deg; joints [3.288, -117.375, -111.913, -40.712, 90, 3.288] of FAIRINO FR5
    - target Target_208 (Cartesian target) at (100, -70, 0) mm, rotated rx -180 ry 0 rz -90 deg; joints [3.348, -116.42, -113.586, -39.994, 90, 3.348] of FAIRINO FR5
    - target Target_209 (Cartesian target) at (90, -70, 0) mm, rotated rx -180 ry 0 rz -90 deg; joints [3.41, -115.466, -115.243, -39.291, 90, 3.41] of FAIRINO FR5
    - target Target_210 (Cartesian target) at (80, -70, 0) mm, rotated rx -180 ry 0 rz -90 deg; joints [3.475, -114.514, -116.884, -38.602, 90, 3.475] of FAIRINO FR5
    - target Target_211 (Cartesian target) at (70, -70, 0) mm, rotated rx -180 ry 0 rz -90 deg; joints [3.543, -113.561, -118.511, -37.928, 90, 3.543] of FAIRINO FR5
    - target Target_212 (Cartesian target) at (60, -70, 0) mm, rotated rx -180 ry 0 rz -90 deg; joints [3.613, -112.608, -120.123, -37.269, 90, 3.613] of FAIRINO FR5
    - target Target_213 (Cartesian target) at (50, -70, 0) mm, rotated rx -180 ry 0 rz -90 deg; joints [3.686, -111.653, -121.722, -36.625, 90, 3.686] of FAIRINO FR5
    - target Target_214 (Cartesian target) at (40, -70, 0) mm, rotated rx -180 ry 0 rz -90 deg; joints [3.762, -110.695, -123.308, -35.997, 90, 3.762] of FAIRINO FR5
    - target Target_215 (Cartesian target) at (30, -70, 0) mm, rotated rx -180 ry 0 rz -90 deg; joints [3.841, -109.734, -124.882, -35.384, 90, 3.841] of FAIRINO FR5
    - target Target_216 (Cartesian target) at (20, -70, 0) mm, rotated rx -180 ry 0 rz -90 deg; joints [3.924, -108.769, -126.443, -34.788, 90, 3.924] of FAIRINO FR5
    - target Target_217 (Cartesian target) at (10, -70, 0) mm, rotated rx -180 ry 0 rz -90 deg; joints [4.01, -107.797, -127.993, -34.209, 90, 4.01] of FAIRINO FR5
    - target Target_218 (Cartesian target) at (0, -70, 0) mm, rotated rx -180 ry 0 rz -90 deg; joints [4.101, -106.819, -129.532, -33.648, 90, 4.101] of FAIRINO FR5
    - target Target_219 (Cartesian target) at (-10, -70, 0) mm, rotated rx -180 ry 0 rz -90 deg; joints [4.195, -105.833, -131.061, -33.106, 90, 4.195] of FAIRINO FR5
    - target Target_220 (Cartesian target) at (-20, -70, 0) mm, rotated rx -180 ry 0 rz -90 deg; joints [4.294, -104.837, -132.579, -32.584, 90, 4.294] of FAIRINO FR5
    - target Target_221 (Cartesian target) at (-30, -70, 0) mm, rotated rx -180 ry 0 rz -90 deg; joints [4.398, -103.831, -134.087, -32.082, 90, 4.398] of FAIRINO FR5
    - target Target_222 (Cartesian target) at (-40, -70, 0) mm, rotated rx -180 ry 0 rz -90 deg; joints [4.507, -102.811, -135.586, -31.603, 90, 4.507] of FAIRINO FR5
    - target Target_223 (Cartesian target) at (-50, -70, 0) mm, rotated rx -180 ry 0 rz -90 deg; joints [4.621, -101.777, -137.075, -31.148, 90, 4.621] of FAIRINO FR5
    - target Target_224 (Cartesian target) at (-60, -70, 0) mm, rotated rx -180 ry 0 rz -90 deg; joints [4.742, -100.726, -138.554, -30.719, 90, 4.742] of FAIRINO FR5
    - target Target_225 (Cartesian target) at (-70, -70, 0) mm, rotated rx -180 ry 0 rz -90 deg; joints [4.869, -99.657, -140.025, -30.318, 90, 4.869] of FAIRINO FR5
    - target Target_226 (Cartesian target) at (-80, -70, 0) mm, rotated rx -180 ry 0 rz -90 deg; joints [5.003, -98.565, -141.487, -29.948, 90, 5.003] of FAIRINO FR5
    - target Target_227 (Cartesian target) at (-90, -70, 0) mm, rotated rx -180 ry 0 rz -90 deg; joints [5.145, -97.449, -142.94, -29.611, 90, 5.145] of FAIRINO FR5
    - target Target_228 (Cartesian target) at (-100, -70, 0) mm, rotated rx -180 ry 0 rz -90 deg; joints [5.295, -96.305, -144.384, -29.311, 90, 5.295] of FAIRINO FR5
    - target Target_229 (Cartesian target) at (-110, -70, 0) mm, rotated rx -180 ry 0 rz -90 deg; joints [5.454, -95.128, -145.819, -29.053, 90, 5.454] of FAIRINO FR5
    - target Target_230 (Cartesian target) at (-120, -70, 0) mm, rotated rx -180 ry 0 rz -90 deg; joints [5.623, -93.915, -147.245, -28.84, 90, 5.623] of FAIRINO FR5
    - target Target_231 (Cartesian target) at (-130, -70, 0) mm, rotated rx -180 ry 0 rz -90 deg; joints [5.804, -92.659, -148.662, -28.679, 90, 5.804] of FAIRINO FR5
    - target Target_232 (Cartesian target) at (-140, -70, 0) mm, rotated rx -180 ry 0 rz -90 deg; joints [5.996, -91.355, -150.068, -28.576, 90, 5.996] of FAIRINO FR5
    - target Target_233 (Cartesian target) at (-140, -60, 0) mm, rotated rx -180 ry 0 rz -90 deg; joints [7.893, -91.074, -150.363, -28.563, 90, 7.893] of FAIRINO FR5
    - target Target_234 (Cartesian target) at (-130, -60, 0) mm, rotated rx -180 ry 0 rz -90 deg; joints [7.638, -92.398, -148.949, -28.653, 90, 7.638] of FAIRINO FR5
    - target Target_235 (Cartesian target) at (-120, -60, 0) mm, rotated rx -180 ry 0 rz -90 deg; joints [7.399, -93.671, -147.526, -28.804, 90, 7.399] of FAIRINO FR5
    - target Target_236 (Cartesian target) at (-110, -60, 0) mm, rotated rx -180 ry 0 rz -90 deg; joints [7.176, -94.899, -146.093, -29.008, 90, 7.176] of FAIRINO FR5
    - target Target_237 (Cartesian target) at (-100, -60, 0) mm, rotated rx -180 ry 0 rz -90 deg; joints [6.965, -96.088, -144.652, -29.26, 90, 6.965] of FAIRINO FR5
    - target Target_238 (Cartesian target) at (-90, -60, 0) mm, rotated rx -180 ry 0 rz -90 deg; joints [6.767, -97.244, -143.202, -29.554, 90, 6.767] of FAIRINO FR5
    - target Target_239 (Cartesian target) at (-80, -60, 0) mm, rotated rx -180 ry 0 rz -90 deg; joints [6.579, -98.371, -141.743, -29.886, 90, 6.579] of FAIRINO FR5
    - target Target_240 (Cartesian target) at (-70, -60, 0) mm, rotated rx -180 ry 0 rz -90 deg; joints [6.402, -99.471, -140.276, -30.252, 90, 6.402] of FAIRINO FR5
    - target Target_241 (Cartesian target) at (-60, -60, 0) mm, rotated rx -180 ry 0 rz -90 deg; joints [6.235, -100.549, -138.801, -30.65, 90, 6.235] of FAIRINO FR5
    - target Target_242 (Cartesian target) at (-50, -60, 0) mm, rotated rx -180 ry 0 rz -90 deg; joints [6.076, -101.607, -137.316, -31.077, 90, 6.076] of FAIRINO FR5
    - target Target_243 (Cartesian target) at (-40, -60, 0) mm, rotated rx -180 ry 0 rz -90 deg; joints [5.925, -102.648, -135.823, -31.529, 90, 5.925] of FAIRINO FR5
    - target Target_244 (Cartesian target) at (-30, -60, 0) mm, rotated rx -180 ry 0 rz -90 deg; joints [5.781, -103.673, -134.32, -32.007, 90, 5.781] of FAIRINO FR5
    - target Target_245 (Cartesian target) at (-20, -60, 0) mm, rotated rx -180 ry 0 rz -90 deg; joints [5.644, -104.686, -132.808, -32.506, 90, 5.644] of FAIRINO FR5
    - target Target_246 (Cartesian target) at (-10, -60, 0) mm, rotated rx -180 ry 0 rz -90 deg; joints [5.514, -105.686, -131.286, -33.028, 90, 5.514] of FAIRINO FR5
    - target Target_247 (Cartesian target) at (0, -60, 0) mm, rotated rx -180 ry 0 rz -90 deg; joints [5.389, -106.677, -129.754, -33.569, 90, 5.389] of FAIRINO FR5
    - target Target_248 (Cartesian target) at (10, -60, 0) mm, rotated rx -180 ry 0 rz -90 deg; joints [5.27, -107.659, -128.212, -34.129, 90, 5.27] of FAIRINO FR5
    - target Target_249 (Cartesian target) at (20, -60, 0) mm, rotated rx -180 ry 0 rz -90 deg; joints [5.157, -108.635, -126.659, -34.707, 90, 5.157] of FAIRINO FR5
    - target Target_250 (Cartesian target) at (30, -60, 0) mm, rotated rx -180 ry 0 rz -90 deg; joints [5.048, -109.604, -125.094, -35.302, 90, 5.048] of FAIRINO FR5
    - target Target_251 (Cartesian target) at (40, -60, 0) mm, rotated rx -180 ry 0 rz -90 deg; joints [4.943, -110.568, -123.518, -35.914, 90, 4.943] of FAIRINO FR5
    - target Target_252 (Cartesian target) at (50, -60, 0) mm, rotated rx -180 ry 0 rz -90 deg; joints [4.843, -111.529, -121.929, -36.542, 90, 4.843] of FAIRINO FR5
    - target Target_253 (Cartesian target) at (60, -60, 0) mm, rotated rx -180 ry 0 rz -90 deg; joints [4.747, -112.486, -120.328, -37.186, 90, 4.747] of FAIRINO FR5
    - target Target_254 (Cartesian target) at (70, -60, 0) mm, rotated rx -180 ry 0 rz -90 deg; joints [4.655, -113.442, -118.713, -37.845, 90, 4.655] of FAIRINO FR5
    - target Target_255 (Cartesian target) at (80, -60, 0) mm, rotated rx -180 ry 0 rz -90 deg; joints [4.566, -114.397, -117.085, -38.519, 90, 4.566] of FAIRINO FR5
    - target Target_256 (Cartesian target) at (90, -60, 0) mm, rotated rx -180 ry 0 rz -90 deg; joints [4.48, -115.352, -115.441, -39.207, 90, 4.48] of FAIRINO FR5
    - target Target_257 (Cartesian target) at (100, -60, 0) mm, rotated rx -180 ry 0 rz -90 deg; joints [4.398, -116.307, -113.783, -39.91, 90, 4.398] of FAIRINO FR5
    - target Target_258 (Cartesian target) at (110, -60, 0) mm, rotated rx -180 ry 0 rz -90 deg; joints [4.319, -117.264, -112.108, -40.628, 90, 4.319] of FAIRINO FR5
    - target Target_259 (Cartesian target) at (120, -60, 0) mm, rotated rx -180 ry 0 rz -90 deg; joints [4.242, -118.223, -110.416, -41.361, 90, 4.242] of FAIRINO FR5
    - target Target_260 (Cartesian target) at (130, -60, 0) mm, rotated rx -180 ry 0 rz -90 deg; joints [4.168, -119.185, -108.707, -42.108, 90, 4.168] of FAIRINO FR5
    - target Target_261 (Cartesian target) at (140, -60, 0) mm, rotated rx -180 ry 0 rz -90 deg; joints [4.097, -120.152, -106.979, -42.87, 90, 4.097] of FAIRINO FR5
    - target Target_262 (Cartesian target) at (140, -50, 0) mm, rotated rx -180 ry 0 rz -90 deg; joints [5.075, -120.061, -107.141, -42.798, 90, 5.075] of FAIRINO FR5
    - target Target_263 (Cartesian target) at (130, -50, 0) mm, rotated rx -180 ry 0 rz -90 deg; joints [5.164, -119.094, -108.87, -42.036, 90, 5.164] of FAIRINO FR5
    - target Target_264 (Cartesian target) at (120, -50, 0) mm, rotated rx -180 ry 0 rz -90 deg; joints [5.255, -118.13, -110.58, -41.289, 90, 5.255] of FAIRINO FR5
    - target Target_265 (Cartesian target) at (110, -50, 0) mm, rotated rx -180 ry 0 rz -90 deg; joints [5.35, -117.17, -112.273, -40.557, 90, 5.35] of FAIRINO FR5
    - target Target_266 (Cartesian target) at (100, -50, 0) mm, rotated rx -180 ry 0 rz -90 deg; joints [5.449, -116.211, -113.949, -39.839, 90, 5.449] of FAIRINO FR5
    - target Target_267 (Cartesian target) at (90, -50, 0) mm, rotated rx -180 ry 0 rz -90 deg; joints [5.551, -115.254, -115.609, -39.136, 90, 5.551] of FAIRINO FR5
    - target Target_268 (Cartesian target) at (80, -50, 0) mm, rotated rx -180 ry 0 rz -90 deg; joints [5.657, -114.298, -117.254, -38.448, 90, 5.657] of FAIRINO FR5
    - target Target_269 (Cartesian target) at (70, -50, 0) mm, rotated rx -180 ry 0 rz -90 deg; joints [5.767, -113.341, -118.885, -37.774, 90, 5.767] of FAIRINO FR5
    - target Target_270 (Cartesian target) at (60, -50, 0) mm, rotated rx -180 ry 0 rz -90 deg; joints [5.882, -112.383, -120.501, -37.116, 90, 5.882] of FAIRINO FR5
    - target Target_271 (Cartesian target) at (50, -50, 0) mm, rotated rx -180 ry 0 rz -90 deg; joints [6.001, -111.423, -122.105, -36.472, 90, 6.001] of FAIRINO FR5
    - target Target_272 (Cartesian target) at (40, -50, 0) mm, rotated rx -180 ry 0 rz -90 deg; joints [6.125, -110.46, -123.695, -35.845, 90, 6.125] of FAIRINO FR5
    - target Target_273 (Cartesian target) at (30, -50, 0) mm, rotated rx -180 ry 0 rz -90 deg; joints [6.255, -109.493, -125.274, -35.233, 90, 6.255] of FAIRINO FR5
    - target Target_274 (Cartesian target) at (20, -50, 0) mm, rotated rx -180 ry 0 rz -90 deg; joints [6.39, -108.521, -126.841, -34.638, 90, 6.39] of FAIRINO FR5
    - target Target_275 (Cartesian target) at (10, -50, 0) mm, rotated rx -180 ry 0 rz -90 deg; joints [6.531, -107.542, -128.397, -34.061, 90, 6.531] of FAIRINO FR5
    - target Target_276 (Cartesian target) at (0, -50, 0) mm, rotated rx -180 ry 0 rz -90 deg; joints [6.679, -106.556, -129.942, -33.501, 90, 6.679] of FAIRINO FR5
    - target Target_277 (Cartesian target) at (-10, -50, 0) mm, rotated rx -180 ry 0 rz -90 deg; joints [6.834, -105.562, -131.477, -32.961, 90, 6.834] of FAIRINO FR5
    - target Target_278 (Cartesian target) at (-20, -50, 0) mm, rotated rx -180 ry 0 rz -90 deg; joints [6.996, -104.557, -133.002, -32.441, 90, 6.996] of FAIRINO FR5
    - target Target_279 (Cartesian target) at (-30, -50, 0) mm, rotated rx -180 ry 0 rz -90 deg; joints [7.166, -103.54, -134.518, -31.943, 90, 7.166] of FAIRINO FR5
    - target Target_280 (Cartesian target) at (-40, -50, 0) mm, rotated rx -180 ry 0 rz -90 deg; joints [7.344, -102.509, -136.024, -31.467, 90, 7.344] of FAIRINO FR5
    - target Target_281 (Cartesian target) at (-50, -50, 0) mm, rotated rx -180 ry 0 rz -90 deg; joints [7.532, -101.463, -137.521, -31.016, 90, 7.532] of FAIRINO FR5
    - target Target_282 (Cartesian target) at (-60, -50, 0) mm, rotated rx -180 ry 0 rz -90 deg; joints [7.73, -100.398, -139.01, -30.592, 90, 7.73] of FAIRINO FR5
    - target Target_283 (Cartesian target) at (-70, -50, 0) mm, rotated rx -180 ry 0 rz -90 deg; joints [7.938, -99.313, -140.49, -30.197, 90, 7.938] of FAIRINO FR5
    - target Target_284 (Cartesian target) at (-80, -50, 0) mm, rotated rx -180 ry 0 rz -90 deg; joints [8.158, -98.205, -141.961, -29.834, 90, 8.158] of FAIRINO FR5
    - target Target_285 (Cartesian target) at (-90, -50, 0) mm, rotated rx -180 ry 0 rz -90 deg; joints [8.391, -97.069, -143.424, -29.506, 90, 8.391] of FAIRINO FR5
    - target Target_286 (Cartesian target) at (-100, -50, 0) mm, rotated rx -180 ry 0 rz -90 deg; joints [8.638, -95.903, -144.879, -29.217, 90, 8.638] of FAIRINO FR5
    - target Target_287 (Cartesian target) at (-110, -50, 0) mm, rotated rx -180 ry 0 rz -90 deg; joints [8.9, -94.702, -146.326, -28.972, 90, 8.9] of FAIRINO FR5
    - target Target_288 (Cartesian target) at (-120, -50, 0) mm, rotated rx -180 ry 0 rz -90 deg; joints [9.179, -93.461, -147.764, -28.775, 90, 9.179] of FAIRINO FR5
    - target Target_289 (Cartesian target) at (-130, -50, 0) mm, rotated rx -180 ry 0 rz -90 deg; joints [9.476, -92.174, -149.193, -28.633, 90, 9.476] of FAIRINO FR5
    - target Target_290 (Cartesian target) at (-140, -50, 0) mm, rotated rx -180 ry 0 rz -90 deg; joints [9.793, -90.832, -150.614, -28.554, 90, 9.793] of FAIRINO FR5
    - target Target_291 (Cartesian target) at (-140, -40, 0) mm, rotated rx -180 ry 0 rz -90 deg; joints [11.694, -90.632, -150.82, -28.548, 90, 11.694] of FAIRINO FR5
    - target Target_292 (Cartesian target) at (-130, -40, 0) mm, rotated rx -180 ry 0 rz -90 deg; joints [11.314, -91.988, -149.394, -28.618, 90, 11.314] of FAIRINO FR5
    - target Target_293 (Cartesian target) at (-120, -40, 0) mm, rotated rx -180 ry 0 rz -90 deg; joints [10.958, -93.288, -147.96, -28.752, 90, 10.958] of FAIRINO FR5
    - target Target_294 (Cartesian target) at (-110, -40, 0) mm, rotated rx -180 ry 0 rz -90 deg; joints [10.624, -94.54, -146.517, -28.943, 90, 10.624] of FAIRINO FR5
    - target Target_295 (Cartesian target) at (-100, -40, 0) mm, rotated rx -180 ry 0 rz -90 deg; joints [10.311, -95.751, -145.066, -29.183, 90, 10.311] of FAIRINO FR5
    - target Target_296 (Cartesian target) at (-90, -40, 0) mm, rotated rx -180 ry 0 rz -90 deg; joints [10.016, -96.925, -143.607, -29.468, 90, 10.016] of FAIRINO FR5
    - target Target_297 (Cartesian target) at (-80, -40, 0) mm, rotated rx -180 ry 0 rz -90 deg; joints [9.737, -98.068, -142.14, -29.792, 90, 9.737] of FAIRINO FR5
    - target Target_298 (Cartesian target) at (-70, -40, 0) mm, rotated rx -180 ry 0 rz -90 deg; joints [9.474, -99.183, -140.665, -30.152, 90, 9.474] of FAIRINO FR5
    - target Target_299 (Cartesian target) at (-60, -40, 0) mm, rotated rx -180 ry 0 rz -90 deg; joints [9.224, -100.274, -139.181, -30.545, 90, 9.224] of FAIRINO FR5
    - target Target_300 (Cartesian target) at (-50, -40, 0) mm, rotated rx -180 ry 0 rz -90 deg; joints [8.988, -101.344, -137.689, -30.967, 90, 8.988] of FAIRINO FR5
    - target Target_301 (Cartesian target) at (-40, -40, 0) mm, rotated rx -180 ry 0 rz -90 deg; joints [8.764, -102.395, -136.189, -31.416, 90, 8.764] of FAIRINO FR5
    - target Target_302 (Cartesian target) at (-30, -40, 0) mm, rotated rx -180 ry 0 rz -90 deg; joints [8.55, -103.43, -134.68, -31.89, 90, 8.55] of FAIRINO FR5
    - target Target_303 (Cartesian target) at (-20, -40, 0) mm, rotated rx -180 ry 0 rz -90 deg; joints [8.347, -104.451, -133.161, -32.388, 90, 8.347] of FAIRINO FR5
    - target Target_304 (Cartesian target) at (-10, -40, 0) mm, rotated rx -180 ry 0 rz -90 deg; joints [8.154, -105.459, -131.634, -32.907, 90, 8.154] of FAIRINO FR5
    - target Target_305 (Cartesian target) at (0, -40, 0) mm, rotated rx -180 ry 0 rz -90 deg; joints [7.969, -106.457, -130.096, -33.446, 90, 7.969] of FAIRINO FR5
    - target Target_306 (Cartesian target) at (10, -40, 0) mm, rotated rx -180 ry 0 rz -90 deg; joints [7.792, -107.446, -128.549, -34.005, 90, 7.792] of FAIRINO FR5
    - target Target_307 (Cartesian target) at (20, -40, 0) mm, rotated rx -180 ry 0 rz -90 deg; joints [7.624, -108.427, -126.991, -34.582, 90, 7.624] of FAIRINO FR5
    - target Target_308 (Cartesian target) at (30, -40, 0) mm, rotated rx -180 ry 0 rz -90 deg; joints [7.462, -109.402, -125.422, -35.177, 90, 7.462] of FAIRINO FR5
    - target Target_309 (Cartesian target) at (40, -40, 0) mm, rotated rx -180 ry 0 rz -90 deg; joints [7.307, -110.371, -123.841, -35.788, 90, 7.307] of FAIRINO FR5
    - target Target_310 (Cartesian target) at (50, -40, 0) mm, rotated rx -180 ry 0 rz -90 deg; joints [7.159, -111.336, -122.249, -36.415, 90, 7.159] of FAIRINO FR5
    - target Target_311 (Cartesian target) at (60, -40, 0) mm, rotated rx -180 ry 0 rz -90 deg; joints [7.017, -112.298, -120.644, -37.058, 90, 7.017] of FAIRINO FR5
    - target Target_312 (Cartesian target) at (70, -40, 0) mm, rotated rx -180 ry 0 rz -90 deg; joints [6.88, -113.258, -119.025, -37.717, 90, 6.88] of FAIRINO FR5
    - target Target_313 (Cartesian target) at (80, -40, 0) mm, rotated rx -180 ry 0 rz -90 deg; joints [6.748, -114.216, -117.393, -38.39, 90, 6.748] of FAIRINO FR5
    - target Target_314 (Cartesian target) at (90, -40, 0) mm, rotated rx -180 ry 0 rz -90 deg; joints [6.621, -115.174, -115.747, -39.078, 90, 6.621] of FAIRINO FR5
    - target Target_315 (Cartesian target) at (100, -40, 0) mm, rotated rx -180 ry 0 rz -90 deg; joints [6.5, -116.133, -114.086, -39.781, 90, 6.5] of FAIRINO FR5
    - target Target_316 (Cartesian target) at (110, -40, 0) mm, rotated rx -180 ry 0 rz -90 deg; joints [6.382, -117.093, -112.409, -40.499, 90, 6.382] of FAIRINO FR5
    - target Target_317 (Cartesian target) at (120, -40, 0) mm, rotated rx -180 ry 0 rz -90 deg; joints [6.269, -118.054, -110.715, -41.231, 90, 6.269] of FAIRINO FR5
    - target Target_318 (Cartesian target) at (130, -40, 0) mm, rotated rx -180 ry 0 rz -90 deg; joints [6.159, -119.019, -109.003, -41.978, 90, 6.159] of FAIRINO FR5
    - target Target_319 (Cartesian target) at (140, -40, 0) mm, rotated rx -180 ry 0 rz -90 deg; joints [6.054, -119.987, -107.273, -42.739, 90, 6.054] of FAIRINO FR5
    - target Target_320 (Cartesian target) at (140, -30, 0) mm, rotated rx -180 ry 0 rz -90 deg; joints [7.032, -119.93, -107.377, -42.694, 90, 7.032] of FAIRINO FR5
    - target Target_321 (Cartesian target) at (130, -30, 0) mm, rotated rx -180 ry 0 rz -90 deg; joints [7.154, -118.961, -109.107, -41.932, 90, 7.154] of FAIRINO FR5
    - target Target_322 (Cartesian target) at (120, -30, 0) mm, rotated rx -180 ry 0 rz -90 deg; joints [7.281, -117.995, -110.819, -41.186, 90, 7.281] of FAIRINO FR5
    - target Target_323 (Cartesian target) at (110, -30, 0) mm, rotated rx -180 ry 0 rz -90 deg; joints [7.413, -117.032, -112.514, -40.454, 90, 7.413] of FAIRINO FR5
    - target Target_324 (Cartesian target) at (100, -30, 0) mm, rotated rx -180 ry 0 rz -90 deg; joints [7.549, -116.072, -114.192, -39.736, 90, 7.549] of FAIRINO FR5
    - target Target_325 (Cartesian target) at (90, -30, 0) mm, rotated rx -180 ry 0 rz -90 deg; joints [7.691, -115.112, -115.854, -39.033, 90, 7.691] of FAIRINO FR5
    - target Target_326 (Cartesian target) at (80, -30, 0) mm, rotated rx -180 ry 0 rz -90 deg; joints [7.838, -114.153, -117.502, -38.345, 90, 7.838] of FAIRINO FR5
    - target Target_327 (Cartesian target) at (70, -30, 0) mm, rotated rx -180 ry 0 rz -90 deg; joints [7.991, -113.193, -119.135, -37.672, 90, 7.991] of FAIRINO FR5
    - target Target_328 (Cartesian target) at (60, -30, 0) mm, rotated rx -180 ry 0 rz -90 deg; joints [8.15, -112.232, -120.754, -37.014, 90, 8.15] of FAIRINO FR5
    - target Target_329 (Cartesian target) at (50, -30, 0) mm, rotated rx -180 ry 0 rz -90 deg; joints [8.316, -111.269, -122.361, -36.371, 90, 8.316] of FAIRINO FR5
    - target Target_330 (Cartesian target) at (40, -30, 0) mm, rotated rx -180 ry 0 rz -90 deg; joints [8.488, -110.302, -123.954, -35.744, 90, 8.488] of FAIRINO FR5
    - target Target_331 (Cartesian target) at (30, -30, 0) mm, rotated rx -180 ry 0 rz -90 deg; joints [8.668, -109.331, -125.537, -35.133, 90, 8.668] of FAIRINO FR5
    - target Target_332 (Cartesian target) at (20, -30, 0) mm, rotated rx -180 ry 0 rz -90 deg; joints [8.856, -108.354, -127.107, -34.539, 90, 8.856] of FAIRINO FR5
    - target Target_333 (Cartesian target) at (10, -30, 0) mm, rotated rx -180 ry 0 rz -90 deg; joints [9.052, -107.371, -128.667, -33.962, 90, 9.052] of FAIRINO FR5
    - target Target_334 (Cartesian target) at (0, -30, 0) mm, rotated rx -180 ry 0 rz -90 deg; joints [9.257, -106.38, -130.216, -33.404, 90, 9.257] of FAIRINO FR5
    - target Target_335 (Cartesian target) at (-10, -30, 0) mm, rotated rx -180 ry 0 rz -90 deg; joints [9.472, -105.379, -131.756, -32.865, 90, 9.472] of FAIRINO FR5
    - target Target_336 (Cartesian target) at (-20, -30, 0) mm, rotated rx -180 ry 0 rz -90 deg; joints [9.697, -104.368, -133.286, -32.347, 90, 9.697] of FAIRINO FR5
    - target Target_337 (Cartesian target) at (-30, -30, 0) mm, rotated rx -180 ry 0 rz -90 deg; joints [9.933, -103.344, -134.806, -31.85, 90, 9.933] of FAIRINO FR5
    - target Target_338 (Cartesian target) at (-40, -30, 0) mm, rotated rx -180 ry 0 rz -90 deg; joints [10.181, -102.306, -136.318, -31.377, 90, 10.181] of FAIRINO FR5
    - target Target_339 (Cartesian target) at (-50, -30, 0) mm, rotated rx -180 ry 0 rz -90 deg; joints [10.442, -101.251, -137.82, -30.929, 90, 10.442] of FAIRINO FR5
    - target Target_340 (Cartesian target) at (-60, -30, 0) mm, rotated rx -180 ry 0 rz -90 deg; joints [10.717, -100.177, -139.315, -30.509, 90, 10.717] of FAIRINO FR5
    - target Target_341 (Cartesian target) at (-70, -30, 0) mm, rotated rx -180 ry 0 rz -90 deg; joints [11.007, -99.081, -140.801, -30.118, 90, 11.007] of FAIRINO FR5
    - target Target_342 (Cartesian target) at (-80, -30, 0) mm, rotated rx -180 ry 0 rz -90 deg; joints [11.313, -97.961, -142.279, -29.76, 90, 11.313] of FAIRINO FR5
    - target Target_343 (Cartesian target) at (-90, -30, 0) mm, rotated rx -180 ry 0 rz -90 deg; joints [11.637, -96.812, -143.749, -29.438, 90, 11.637] of FAIRINO FR5
    - target Target_344 (Cartesian target) at (-100, -30, 0) mm, rotated rx -180 ry 0 rz -90 deg; joints [11.981, -95.631, -145.212, -29.157, 90, 11.981] of FAIRINO FR5
    - target Target_345 (Cartesian target) at (-110, -30, 0) mm, rotated rx -180 ry 0 rz -90 deg; joints [12.345, -94.413, -146.666, -28.921, 90, 12.345] of FAIRINO FR5
    - target Target_346 (Cartesian target) at (-120, -30, 0) mm, rotated rx -180 ry 0 rz -90 deg; joints [12.734, -93.152, -148.113, -28.735, 90, 12.734] of FAIRINO FR5
    - target Target_347 (Cartesian target) at (-130, -30, 0) mm, rotated rx -180 ry 0 rz -90 deg; joints [13.147, -91.842, -149.551, -28.607, 90, 13.147] of FAIRINO FR5
    - target Target_348 (Cartesian target) at (-140, -30, 0) mm, rotated rx -180 ry 0 rz -90 deg; joints [13.59, -90.475, -150.98, -28.545, 90, 13.59] of FAIRINO FR5
    - target Target_349 (Cartesian target) at (-140, -20, 0) mm, rotated rx -180 ry 0 rz -90 deg; joints [15.477, -90.362, -151.095, -28.543, 90, 15.477] of FAIRINO FR5
    - target Target_350 (Cartesian target) at (-130, -20, 0) mm, rotated rx -180 ry 0 rz -90 deg; joints [14.973, -91.738, -149.663, -28.6, 90, 14.973] of FAIRINO FR5
    - target Target_351 (Cartesian target) at (-120, -20, 0) mm, rotated rx -180 ry 0 rz -90 deg; joints [14.502, -93.055, -148.222, -28.723, 90, 14.502] of FAIRINO FR5
    - target Target_352 (Cartesian target) at (-110, -20, 0) mm, rotated rx -180 ry 0 rz -90 deg; joints [14.06, -94.322, -146.773, -28.905, 90, 14.06] of FAIRINO FR5
    - target Target_353 (Cartesian target) at (-100, -20, 0) mm, rotated rx -180 ry 0 rz -90 deg; joints [13.645, -95.545, -145.316, -29.138, 90, 13.645] of FAIRINO FR5
    - target Target_354 (Cartesian target) at (-90, -20, 0) mm, rotated rx -180 ry 0 rz -90 deg; joints [13.253, -96.731, -143.851, -29.417, 90, 13.253] of FAIRINO FR5
    - target Target_355 (Cartesian target) at (-80, -20, 0) mm, rotated rx -180 ry 0 rz -90 deg; joints [12.884, -97.884, -142.379, -29.737, 90, 12.884] of FAIRINO FR5
    - target Target_356 (Cartesian target) at (-70, -20, 0) mm, rotated rx -180 ry 0 rz -90 deg; joints [12.535, -99.008, -140.899, -30.093, 90, 12.535] of FAIRINO FR5
    - target Target_357 (Cartesian target) at (-60, -20, 0) mm, rotated rx -180 ry 0 rz -90 deg; joints [12.205, -100.107, -139.41, -30.483, 90, 12.205] of FAIRINO FR5
    - target Target_358 (Cartesian target) at (-50, -20, 0) mm, rotated rx -180 ry 0 rz -90 deg; joints [11.892, -101.184, -137.914, -30.902, 90, 11.892] of FAIRINO FR5
    - target Target_359 (Cartesian target) at (-40, -20, 0) mm, rotated rx -180 ry 0 rz -90 deg; joints [11.595, -102.242, -136.409, -31.349, 90, 11.595] of FAIRINO FR5
    - target Target_360 (Cartesian target) at (-30, -20, 0) mm, rotated rx -180 ry 0 rz -90 deg; joints [11.313, -103.283, -134.896, -31.821, 90, 11.313] of FAIRINO FR5
    - target Target_361 (Cartesian target) at (-20, -20, 0) mm, rotated rx -180 ry 0 rz -90 deg; joints [11.044, -104.309, -133.374, -32.317, 90, 11.044] of FAIRINO FR5
    - target Target_362 (Cartesian target) at (-10, -20, 0) mm, rotated rx -180 ry 0 rz -90 deg; joints [10.787, -105.322, -131.843, -32.835, 90, 10.787] of FAIRINO FR5
    - target Target_363 (Cartesian target) at (0, -20, 0) mm, rotated rx -180 ry 0 rz -90 deg; joints [10.543, -106.324, -130.302, -33.373, 90, 10.543] of FAIRINO FR5
    - target Target_364 (Cartesian target) at (10, -20, 0) mm, rotated rx -180 ry 0 rz -90 deg; joints [10.309, -107.317, -128.752, -33.931, 90, 10.309] of FAIRINO FR5
    - target Target_365 (Cartesian target) at (20, -20, 0) mm, rotated rx -180 ry 0 rz -90 deg; joints [10.086, -108.302, -127.19, -34.507, 90, 10.086] of FAIRINO FR5
    - target Target_366 (Cartesian target) at (30, -20, 0) mm, rotated rx -180 ry 0 rz -90 deg; joints [9.872, -109.28, -125.619, -35.101, 90, 9.872] of FAIRINO FR5
    - target Target_367 (Cartesian target) at (40, -20, 0) mm, rotated rx -180 ry 0 rz -90 deg; joints [9.667, -110.253, -124.035, -35.712, 90, 9.667] of FAIRINO FR5
    - target Target_368 (Cartesian target) at (50, -20, 0) mm, rotated rx -180 ry 0 rz -90 deg; joints [9.471, -111.221, -122.441, -36.339, 90, 9.471] of FAIRINO FR5
    - target Target_369 (Cartesian target) at (60, -20, 0) mm, rotated rx -180 ry 0 rz -90 deg; joints [9.282, -112.185, -120.833, -36.982, 90, 9.282] of FAIRINO FR5
    - target Target_370 (Cartesian target) at (70, -20, 0) mm, rotated rx -180 ry 0 rz -90 deg; joints [9.101, -113.147, -119.213, -37.64, 90, 9.101] of FAIRINO FR5
    - target Target_371 (Cartesian target) at (80, -20, 0) mm, rotated rx -180 ry 0 rz -90 deg; joints [8.927, -114.108, -117.579, -38.313, 90, 8.927] of FAIRINO FR5
    - target Target_372 (Cartesian target) at (90, -20, 0) mm, rotated rx -180 ry 0 rz -90 deg; joints [8.759, -115.068, -115.931, -39.001, 90, 8.759] of FAIRINO FR5
    - target Target_373 (Cartesian target) at (100, -20, 0) mm, rotated rx -180 ry 0 rz -90 deg; joints [8.598, -116.028, -114.268, -39.704, 90, 8.598] of FAIRINO FR5
    - target Target_374 (Cartesian target) at (110, -20, 0) mm, rotated rx -180 ry 0 rz -90 deg; joints [8.442, -116.99, -112.589, -40.421, 90, 8.442] of FAIRINO FR5
    - target Target_375 (Cartesian target) at (120, -20, 0) mm, rotated rx -180 ry 0 rz -90 deg; joints [8.292, -117.953, -110.894, -41.153, 90, 8.292] of FAIRINO FR5
    - target Target_376 (Cartesian target) at (130, -20, 0) mm, rotated rx -180 ry 0 rz -90 deg; joints [8.148, -118.919, -109.181, -41.9, 90, 8.148] of FAIRINO FR5
    - target Target_377 (Cartesian target) at (140, -20, 0) mm, rotated rx -180 ry 0 rz -90 deg; joints [8.008, -119.889, -107.45, -42.661, 90, 8.008] of FAIRINO FR5
    - target Target_378 (Cartesian target) at (140, -10, 0) mm, rotated rx -180 ry 0 rz -90 deg; joints [8.983, -119.864, -107.495, -42.642, 90, 8.983] of FAIRINO FR5
    - target Target_379 (Cartesian target) at (130, -10, 0) mm, rotated rx -180 ry 0 rz -90 deg; joints [9.14, -118.894, -109.226, -41.88, 90, 9.14] of FAIRINO FR5
    - target Target_380 (Cartesian target) at (120, -10, 0) mm, rotated rx -180 ry 0 rz -90 deg; joints [9.302, -117.928, -110.939, -41.134, 90, 9.302] of FAIRINO FR5
    - target Target_381 (Cartesian target) at (110, -10, 0) mm, rotated rx -180 ry 0 rz -90 deg; joints [9.47, -116.964, -112.634, -40.402, 90, 9.47] of FAIRINO FR5
    - target Target_382 (Cartesian target) at (100, -10, 0) mm, rotated rx -180 ry 0 rz -90 deg; joints [9.644, -116.002, -114.314, -39.684, 90, 9.644] of FAIRINO FR5
    - target Target_383 (Cartesian target) at (90, -10, 0) mm, rotated rx -180 ry 0 rz -90 deg; joints [9.825, -115.041, -115.977, -38.982, 90, 9.825] of FAIRINO FR5
    - target Target_384 (Cartesian target) at (80, -10, 0) mm, rotated rx -180 ry 0 rz -90 deg; joints [10.013, -114.081, -117.626, -38.294, 90, 10.013] of FAIRINO FR5
    - target Target_385 (Cartesian target) at (70, -10, 0) mm, rotated rx -180 ry 0 rz -90 deg; joints [10.208, -113.119, -119.26, -37.621, 90, 10.208] of FAIRINO FR5
    - target Target_386 (Cartesian target) at (60, -10, 0) mm, rotated rx -180 ry 0 rz -90 deg; joints [10.411, -112.157, -120.881, -36.963, 90, 10.411] of FAIRINO FR5
    - target Target_387 (Cartesian target) at (50, -10, 0) mm, rotated rx -180 ry 0 rz -90 deg; joints [10.623, -111.192, -122.489, -36.32, 90, 10.623] of FAIRINO FR5
    - target Target_388 (Cartesian target) at (40, -10, 0) mm, rotated rx -180 ry 0 rz -90 deg; joints [10.843, -110.223, -124.084, -35.693, 90, 10.843] of FAIRINO FR5
    - target Target_389 (Cartesian target) at (30, -10, 0) mm, rotated rx -180 ry 0 rz -90 deg; joints [11.073, -109.25, -125.668, -35.082, 90, 11.073] of FAIRINO FR5
    - target Target_390 (Cartesian target) at (20, -10, 0) mm, rotated rx -180 ry 0 rz -90 deg; joints [11.312, -108.271, -127.24, -34.489, 90, 11.312] of FAIRINO FR5
    - target Target_391 (Cartesian target) at (10, -10, 0) mm, rotated rx -180 ry 0 rz -90 deg; joints [11.563, -107.285, -128.802, -33.913, 90, 11.563] of FAIRINO FR5
    - target Target_392 (Cartesian target) at (0, -10, 0) mm, rotated rx -180 ry 0 rz -90 deg; joints [11.825, -106.291, -130.354, -33.355, 90, 11.825] of FAIRINO FR5
    - target Target_393 (Cartesian target) at (-10, -10, 0) mm, rotated rx -180 ry 0 rz -90 deg; joints [12.099, -105.288, -131.895, -32.817, 90, 12.099] of FAIRINO FR5
    - target Target_394 (Cartesian target) at (-20, -10, 0) mm, rotated rx -180 ry 0 rz -90 deg; joints [12.386, -104.273, -133.428, -32.299, 90, 12.386] of FAIRINO FR5
    - target Target_395 (Cartesian target) at (-30, -10, 0) mm, rotated rx -180 ry 0 rz -90 deg; joints [12.687, -103.246, -134.951, -31.804, 90, 12.687] of FAIRINO FR5
    - target Target_396 (Cartesian target) at (-40, -10, 0) mm, rotated rx -180 ry 0 rz -90 deg; joints [13.004, -102.203, -136.465, -31.332, 90, 13.004] of FAIRINO FR5
    - target Target_397 (Cartesian target) at (-50, -10, 0) mm, rotated rx -180 ry 0 rz -90 deg; joints [13.337, -101.144, -137.97, -30.886, 90, 13.337] of FAIRINO FR5
    - target Target_398 (Cartesian target) at (-60, -10, 0) mm, rotated rx -180 ry 0 rz -90 deg; joints [13.687, -100.065, -139.468, -30.467, 90, 13.687] of FAIRINO FR5
    - target Target_399 (Cartesian target) at (-70, -10, 0) mm, rotated rx -180 ry 0 rz -90 deg; joints [14.057, -98.964, -140.957, -30.079, 90, 14.057] of FAIRINO FR5
    - target Target_400 (Cartesian target) at (-80, -10, 0) mm, rotated rx -180 ry 0 rz -90 deg; joints [14.448, -97.838, -142.439, -29.723, 90, 14.448] of FAIRINO FR5
    - target Target_401 (Cartesian target) at (-90, -10, 0) mm, rotated rx -180 ry 0 rz -90 deg; joints [14.862, -96.682, -143.913, -29.405, 90, 14.862] of FAIRINO FR5
    - target Target_402 (Cartesian target) at (-100, -10, 0) mm, rotated rx -180 ry 0 rz -90 deg; joints [15.3, -95.494, -145.379, -29.127, 90, 15.3] of FAIRINO FR5
    - target Target_403 (Cartesian target) at (-110, -10, 0) mm, rotated rx -180 ry 0 rz -90 deg; joints [15.765, -94.267, -146.837, -28.896, 90, 15.765] of FAIRINO FR5
    - target Target_404 (Cartesian target) at (-120, -10, 0) mm, rotated rx -180 ry 0 rz -90 deg; joints [16.26, -92.996, -148.288, -28.716, 90, 16.26] of FAIRINO FR5
    - target Target_405 (Cartesian target) at (-130, -10, 0) mm, rotated rx -180 ry 0 rz -90 deg; joints [16.788, -91.674, -149.73, -28.595, 90, 16.788] of FAIRINO FR5
    - target Target_406 (Cartesian target) at (-140, -10, 0) mm, rotated rx -180 ry 0 rz -90 deg; joints [17.352, -90.294, -151.164, -28.542, 90, 17.352] of FAIRINO FR5
    - target Target_407 (Cartesian target) at (-140, 0, 0) mm, rotated rx -180 ry 0 rz -90 deg; joints [19.21, -90.271, -151.188, -28.542, 90, 19.21] of FAIRINO FR5
    - target Target_408 (Cartesian target) at (-130, 0, 0) mm, rotated rx -180 ry 0 rz -90 deg; joints [18.587, -91.653, -149.753, -28.594, 90, 18.587] of FAIRINO FR5
    - target Target_409 (Cartesian target) at (-120, 0, 0) mm, rotated rx -180 ry 0 rz -90 deg; joints [18.004, -92.976, -148.31, -28.714, 90, 18.004] of FAIRINO FR5
    - target Target_410 (Cartesian target) at (-110, 0, 0) mm, rotated rx -180 ry 0 rz -90 deg; joints [17.458, -94.249, -146.859, -28.893, 90, 17.458] of FAIRINO FR5
    - target Target_411 (Cartesian target) at (-100, 0, 0) mm, rotated rx -180 ry 0 rz -90 deg; joints [16.944, -95.477, -145.4, -29.124, 90, 16.944] of FAIRINO FR5
    - target Target_412 (Cartesian target) at (-90, 0, 0) mm, rotated rx -180 ry 0 rz -90 deg; joints [16.459, -96.666, -143.933, -29.401, 90, 16.459] of FAIRINO FR5
    - target Target_413 (Cartesian target) at (-80, 0, 0) mm, rotated rx -180 ry 0 rz -90 deg; joints [16.002, -97.822, -142.459, -29.719, 90, 16.002] of FAIRINO FR5
    - target Target_414 (Cartesian target) at (-70, 0, 0) mm, rotated rx -180 ry 0 rz -90 deg; joints [15.57, -98.95, -140.977, -30.074, 90, 15.57] of FAIRINO FR5
    - target Target_415 (Cartesian target) at (-60, 0, 0) mm, rotated rx -180 ry 0 rz -90 deg; joints [15.161, -100.051, -139.487, -30.462, 90, 15.161] of FAIRINO FR5
    - target Target_416 (Cartesian target) at (-50, 0, 0) mm, rotated rx -180 ry 0 rz -90 deg; joints [14.774, -101.131, -137.989, -30.88, 90, 14.774] of FAIRINO FR5
    - target Target_417 (Cartesian target) at (-40, 0, 0) mm, rotated rx -180 ry 0 rz -90 deg; joints [14.405, -102.19, -136.483, -31.326, 90, 14.405] of FAIRINO FR5
    - target Target_418 (Cartesian target) at (-30, 0, 0) mm, rotated rx -180 ry 0 rz -90 deg; joints [14.055, -103.233, -134.969, -31.798, 90, 14.055] of FAIRINO FR5
    - target Target_419 (Cartesian target) at (-20, 0, 0) mm, rotated rx -180 ry 0 rz -90 deg; joints [13.722, -104.261, -133.445, -32.293, 90, 13.722] of FAIRINO FR5
    - target Target_420 (Cartesian target) at (-10, 0, 0) mm, rotated rx -180 ry 0 rz -90 deg; joints [13.404, -105.276, -131.913, -32.811, 90, 13.404] of FAIRINO FR5
    - target Target_421 (Cartesian target) at (0, 0, 0) mm, rotated rx -180 ry 0 rz -90 deg; joints [13.101, -106.28, -130.371, -33.349, 90, 13.101] of FAIRINO FR5
    - target Target_422 (Cartesian target) at (10, 0, 0) mm, rotated rx -180 ry 0 rz -90 deg; joints [12.811, -107.274, -128.819, -33.906, 90, 12.811] of FAIRINO FR5
    - target Target_423 (Cartesian target) at (20, 0, 0) mm, rotated rx -180 ry 0 rz -90 deg; joints [12.534, -108.26, -127.257, -34.483, 90, 12.534] of FAIRINO FR5
    - target Target_424 (Cartesian target) at (30, 0, 0) mm, rotated rx -180 ry 0 rz -90 deg; joints [12.269, -109.239, -125.684, -35.076, 90, 12.269] of FAIRINO FR5
    - target Target_425 (Cartesian target) at (40, 0, 0) mm, rotated rx -180 ry 0 rz -90 deg; joints [12.015, -110.213, -124.1, -35.687, 90, 12.015] of FAIRINO FR5
    - target Target_426 (Cartesian target) at (50, 0, 0) mm, rotated rx -180 ry 0 rz -90 deg; joints [11.771, -111.182, -122.505, -36.314, 90, 11.771] of FAIRINO FR5
    - target Target_427 (Cartesian target) at (60, 0, 0) mm, rotated rx -180 ry 0 rz -90 deg; joints [11.537, -112.147, -120.897, -36.956, 90, 11.537] of FAIRINO FR5
    - target Target_428 (Cartesian target) at (70, 0, 0) mm, rotated rx -180 ry 0 rz -90 deg; joints [11.312, -113.11, -119.276, -37.614, 90, 11.312] of FAIRINO FR5
    - target Target_429 (Cartesian target) at (80, 0, 0) mm, rotated rx -180 ry 0 rz -90 deg; joints [11.096, -114.072, -117.641, -38.287, 90, 11.096] of FAIRINO FR5
    - target Target_430 (Cartesian target) at (90, 0, 0) mm, rotated rx -180 ry 0 rz -90 deg; joints [10.888, -115.032, -115.992, -38.975, 90, 10.888] of FAIRINO FR5
    - target Target_431 (Cartesian target) at (100, 0, 0) mm, rotated rx -180 ry 0 rz -90 deg; joints [10.688, -115.993, -114.329, -39.678, 90, 10.688] of FAIRINO FR5
    - target Target_432 (Cartesian target) at (110, 0, 0) mm, rotated rx -180 ry 0 rz -90 deg; joints [10.495, -116.955, -112.65, -40.395, 90, 10.495] of FAIRINO FR5
    - target Target_433 (Cartesian target) at (120, 0, 0) mm, rotated rx -180 ry 0 rz -90 deg; joints [10.308, -117.919, -110.954, -41.127, 90, 10.308] of FAIRINO FR5
    - target Target_434 (Cartesian target) at (130, 0, 0) mm, rotated rx -180 ry 0 rz -90 deg; joints [10.129, -118.886, -109.241, -41.874, 90, 10.129] of FAIRINO FR5
    - target Target_435 (Cartesian target) at (140, 0, 0) mm, rotated rx -180 ry 0 rz -90 deg; joints [9.955, -119.856, -107.509, -42.635, 90, 9.955] of FAIRINO FR5
    - target Target_436 (Cartesian target) at (140, 10, 0) mm, rotated rx -180 ry 0 rz -90 deg; joints [10.925, -119.864, -107.495, -42.642, 90, 10.925] of FAIRINO FR5
    - target Target_437 (Cartesian target) at (130, 10, 0) mm, rotated rx -180 ry 0 rz -90 deg; joints [11.115, -118.894, -109.226, -41.88, 90, 11.115] of FAIRINO FR5
    - target Target_438 (Cartesian target) at (120, 10, 0) mm, rotated rx -180 ry 0 rz -90 deg; joints [11.312, -117.928, -110.939, -41.134, 90, 11.312] of FAIRINO FR5
    - target Target_439 (Cartesian target) at (110, 10, 0) mm, rotated rx -180 ry 0 rz -90 deg; joints [11.516, -116.964, -112.634, -40.402, 90, 11.516] of FAIRINO FR5
    - target Target_440 (Cartesian target) at (100, 10, 0) mm, rotated rx -180 ry 0 rz -90 deg; joints [11.727, -116.002, -114.314, -39.684, 90, 11.727] of FAIRINO FR5
    - target Target_441 (Cartesian target) at (90, 10, 0) mm, rotated rx -180 ry 0 rz -90 deg; joints [11.947, -115.041, -115.977, -38.982, 90, 11.947] of FAIRINO FR5
    - target Target_442 (Cartesian target) at (80, 10, 0) mm, rotated rx -180 ry 0 rz -90 deg; joints [12.175, -114.081, -117.626, -38.294, 90, 12.175] of FAIRINO FR5
    - target Target_443 (Cartesian target) at (70, 10, 0) mm, rotated rx -180 ry 0 rz -90 deg; joints [12.412, -113.119, -119.26, -37.621, 90, 12.412] of FAIRINO FR5
    - target Target_444 (Cartesian target) at (60, 10, 0) mm, rotated rx -180 ry 0 rz -90 deg; joints [12.658, -112.157, -120.881, -36.963, 90, 12.658] of FAIRINO FR5
    - target Target_445 (Cartesian target) at (50, 10, 0) mm, rotated rx -180 ry 0 rz -90 deg; joints [12.914, -111.192, -122.489, -36.32, 90, 12.914] of FAIRINO FR5
    - target Target_446 (Cartesian target) at (40, 10, 0) mm, rotated rx -180 ry 0 rz -90 deg; joints [13.181, -110.223, -124.084, -35.693, 90, 13.181] of FAIRINO FR5
    - target Target_447 (Cartesian target) at (30, 10, 0) mm, rotated rx -180 ry 0 rz -90 deg; joints [13.46, -109.25, -125.668, -35.082, 90, 13.46] of FAIRINO FR5
    - target Target_448 (Cartesian target) at (20, 10, 0) mm, rotated rx -180 ry 0 rz -90 deg; joints [13.75, -108.271, -127.24, -34.489, 90, 13.75] of FAIRINO FR5
    - target Target_449 (Cartesian target) at (10, 10, 0) mm, rotated rx -180 ry 0 rz -90 deg; joints [14.053, -107.285, -128.802, -33.913, 90, 14.053] of FAIRINO FR5
    - target Target_450 (Cartesian target) at (0, 10, 0) mm, rotated rx -180 ry 0 rz -90 deg; joints [14.371, -106.291, -130.354, -33.355, 90, 14.371] of FAIRINO FR5
    - target Target_451 (Cartesian target) at (-10, 10, 0) mm, rotated rx -180 ry 0 rz -90 deg; joints [14.703, -105.288, -131.895, -32.817, 90, 14.703] of FAIRINO FR5
    - target Target_452 (Cartesian target) at (-20, 10, 0) mm, rotated rx -180 ry 0 rz -90 deg; joints [15.05, -104.273, -133.428, -32.299, 90, 15.05] of FAIRINO FR5
    - target Target_453 (Cartesian target) at (-30, 10, 0) mm, rotated rx -180 ry 0 rz -90 deg; joints [15.415, -103.246, -134.951, -31.804, 90, 15.415] of FAIRINO FR5
    - target Target_454 (Cartesian target) at (-40, 10, 0) mm, rotated rx -180 ry 0 rz -90 deg; joints [15.798, -102.203, -136.465, -31.332, 90, 15.798] of FAIRINO FR5
    - target Target_455 (Cartesian target) at (-50, 10, 0) mm, rotated rx -180 ry 0 rz -90 deg; joints [16.201, -101.144, -137.97, -30.886, 90, 16.201] of FAIRINO FR5
    - target Target_456 (Cartesian target) at (-60, 10, 0) mm, rotated rx -180 ry 0 rz -90 deg; joints [16.625, -100.065, -139.468, -30.467, 90, 16.625] of FAIRINO FR5
    - target Target_457 (Cartesian target) at (-70, 10, 0) mm, rotated rx -180 ry 0 rz -90 deg; joints [17.072, -98.964, -140.957, -30.079, 90, 17.072] of FAIRINO FR5
    - target Target_458 (Cartesian target) at (-80, 10, 0) mm, rotated rx -180 ry 0 rz -90 deg; joints [17.544, -97.838, -142.439, -29.723, 90, 17.544] of FAIRINO FR5
    - target Target_459 (Cartesian target) at (-90, 10, 0) mm, rotated rx -180 ry 0 rz -90 deg; joints [18.044, -96.682, -143.913, -29.405, 90, 18.044] of FAIRINO FR5
    - target Target_460 (Cartesian target) at (-100, 10, 0) mm, rotated rx -180 ry 0 rz -90 deg; joints [18.573, -95.494, -145.379, -29.127, 90, 18.573] of FAIRINO FR5
    - target Target_461 (Cartesian target) at (-110, 10, 0) mm, rotated rx -180 ry 0 rz -90 deg; joints [19.134, -94.267, -146.837, -28.896, 90, 19.134] of FAIRINO FR5
    - target Target_462 (Cartesian target) at (-120, 10, 0) mm, rotated rx -180 ry 0 rz -90 deg; joints [19.732, -92.996, -148.288, -28.716, 90, 19.732] of FAIRINO FR5
    - target Target_463 (Cartesian target) at (-130, 10, 0) mm, rotated rx -180 ry 0 rz -90 deg; joints [20.368, -91.674, -149.73, -28.595, 90, 20.368] of FAIRINO FR5
    - target Target_464 (Cartesian target) at (-140, 10, 0) mm, rotated rx -180 ry 0 rz -90 deg; joints [21.047, -90.294, -151.164, -28.542, 90, 21.047] of FAIRINO FR5
    - target Target_465 (Cartesian target) at (-140, 20, 0) mm, rotated rx -180 ry 0 rz -90 deg; joints [22.86, -90.362, -151.095, -28.543, 90, 22.86] of FAIRINO FR5
    - target Target_466 (Cartesian target) at (-130, 20, 0) mm, rotated rx -180 ry 0 rz -90 deg; joints [22.126, -91.738, -149.663, -28.6, 90, 22.126] of FAIRINO FR5
    - target Target_467 (Cartesian target) at (-120, 20, 0) mm, rotated rx -180 ry 0 rz -90 deg; joints [21.439, -93.055, -148.222, -28.723, 90, 21.439] of FAIRINO FR5
    - target Target_468 (Cartesian target) at (-110, 20, 0) mm, rotated rx -180 ry 0 rz -90 deg; joints [20.793, -94.322, -146.773, -28.905, 90, 20.793] of FAIRINO FR5
    - target Target_469 (Cartesian target) at (-100, 20, 0) mm, rotated rx -180 ry 0 rz -90 deg; joints [20.186, -95.545, -145.316, -29.138, 90, 20.186] of FAIRINO FR5
    - target Target_470 (Cartesian target) at (-90, 20, 0) mm, rotated rx -180 ry 0 rz -90 deg; joints [19.613, -96.731, -143.851, -29.417, 90, 19.613] of FAIRINO FR5
    - target Target_471 (Cartesian target) at (-80, 20, 0) mm, rotated rx -180 ry 0 rz -90 deg; joints [19.072, -97.884, -142.379, -29.737, 90, 19.072] of FAIRINO FR5
    - target Target_472 (Cartesian target) at (-70, 20, 0) mm, rotated rx -180 ry 0 rz -90 deg; joints [18.561, -99.008, -140.899, -30.093, 90, 18.561] of FAIRINO FR5
    - target Target_473 (Cartesian target) at (-60, 20, 0) mm, rotated rx -180 ry 0 rz -90 deg; joints [18.077, -100.107, -139.41, -30.483, 90, 18.077] of FAIRINO FR5
    - target Target_474 (Cartesian target) at (-50, 20, 0) mm, rotated rx -180 ry 0 rz -90 deg; joints [17.617, -101.184, -137.914, -30.902, 90, 17.617] of FAIRINO FR5
    - target Target_475 (Cartesian target) at (-40, 20, 0) mm, rotated rx -180 ry 0 rz -90 deg; joints [17.181, -102.242, -136.409, -31.349, 90, 17.181] of FAIRINO FR5
    - target Target_476 (Cartesian target) at (-30, 20, 0) mm, rotated rx -180 ry 0 rz -90 deg; joints [16.765, -103.283, -134.896, -31.821, 90, 16.765] of FAIRINO FR5
    - target Target_477 (Cartesian target) at (-20, 20, 0) mm, rotated rx -180 ry 0 rz -90 deg; joints [16.37, -104.309, -133.374, -32.317, 90, 16.37] of FAIRINO FR5
    - target Target_478 (Cartesian target) at (-10, 20, 0) mm, rotated rx -180 ry 0 rz -90 deg; joints [15.993, -105.322, -131.843, -32.835, 90, 15.993] of FAIRINO FR5
    - target Target_479 (Cartesian target) at (0, 20, 0) mm, rotated rx -180 ry 0 rz -90 deg; joints [15.633, -106.324, -130.302, -33.373, 90, 15.633] of FAIRINO FR5
    - target Target_480 (Cartesian target) at (10, 20, 0) mm, rotated rx -180 ry 0 rz -90 deg; joints [15.288, -107.317, -128.752, -33.931, 90, 15.288] of FAIRINO FR5
    - target Target_481 (Cartesian target) at (20, 20, 0) mm, rotated rx -180 ry 0 rz -90 deg; joints [14.959, -108.302, -127.19, -34.507, 90, 14.959] of FAIRINO FR5
    - target Target_482 (Cartesian target) at (30, 20, 0) mm, rotated rx -180 ry 0 rz -90 deg; joints [14.644, -109.28, -125.619, -35.101, 90, 14.644] of FAIRINO FR5
    - target Target_483 (Cartesian target) at (40, 20, 0) mm, rotated rx -180 ry 0 rz -90 deg; joints [14.342, -110.253, -124.035, -35.712, 90, 14.342] of FAIRINO FR5
    - target Target_484 (Cartesian target) at (50, 20, 0) mm, rotated rx -180 ry 0 rz -90 deg; joints [14.052, -111.221, -122.441, -36.339, 90, 14.052] of FAIRINO FR5
    - target Target_485 (Cartesian target) at (60, 20, 0) mm, rotated rx -180 ry 0 rz -90 deg; joints [13.774, -112.185, -120.833, -36.982, 90, 13.774] of FAIRINO FR5
    - target Target_486 (Cartesian target) at (70, 20, 0) mm, rotated rx -180 ry 0 rz -90 deg; joints [13.506, -113.147, -119.213, -37.64, 90, 13.506] of FAIRINO FR5
    - target Target_487 (Cartesian target) at (80, 20, 0) mm, rotated rx -180 ry 0 rz -90 deg; joints [13.249, -114.108, -117.579, -38.313, 90, 13.249] of FAIRINO FR5
    - target Target_488 (Cartesian target) at (90, 20, 0) mm, rotated rx -180 ry 0 rz -90 deg; joints [13.001, -115.068, -115.931, -39.001, 90, 13.001] of FAIRINO FR5
    - target Target_489 (Cartesian target) at (100, 20, 0) mm, rotated rx -180 ry 0 rz -90 deg; joints [12.763, -116.028, -114.268, -39.704, 90, 12.763] of FAIRINO FR5
    - target Target_490 (Cartesian target) at (110, 20, 0) mm, rotated rx -180 ry 0 rz -90 deg; joints [12.533, -116.99, -112.589, -40.421, 90, 12.533] of FAIRINO FR5
    - target Target_491 (Cartesian target) at (120, 20, 0) mm, rotated rx -180 ry 0 rz -90 deg; joints [12.312, -117.953, -110.894, -41.153, 90, 12.312] of FAIRINO FR5
    - target Target_492 (Cartesian target) at (130, 20, 0) mm, rotated rx -180 ry 0 rz -90 deg; joints [12.098, -118.919, -109.181, -41.9, 90, 12.098] of FAIRINO FR5
    - target Target_493 (Cartesian target) at (140, 20, 0) mm, rotated rx -180 ry 0 rz -90 deg; joints [11.891, -119.889, -107.45, -42.661, 90, 11.891] of FAIRINO FR5
    - target Target_494 (Cartesian target) at (140, 30, 0) mm, rotated rx -180 ry 0 rz -90 deg; joints [12.853, -119.93, -107.377, -42.694, 90, 12.853] of FAIRINO FR5
    - target Target_495 (Cartesian target) at (130, 30, 0) mm, rotated rx -180 ry 0 rz -90 deg; joints [13.076, -118.961, -109.107, -41.932, 90, 13.076] of FAIRINO FR5
    - target Target_496 (Cartesian target) at (120, 30, 0) mm, rotated rx -180 ry 0 rz -90 deg; joints [13.307, -117.995, -110.819, -41.186, 90, 13.307] of FAIRINO FR5
    - target Target_497 (Cartesian target) at (110, 30, 0) mm, rotated rx -180 ry 0 rz -90 deg; joints [13.546, -117.032, -112.514, -40.454, 90, 13.546] of FAIRINO FR5
    - target Target_498 (Cartesian target) at (100, 30, 0) mm, rotated rx -180 ry 0 rz -90 deg; joints [13.794, -116.072, -114.192, -39.736, 90, 13.794] of FAIRINO FR5
    - target Target_499 (Cartesian target) at (90, 30, 0) mm, rotated rx -180 ry 0 rz -90 deg; joints [14.051, -115.112, -115.854, -39.033, 90, 14.051] of FAIRINO FR5
    - target Target_500 (Cartesian target) at (80, 30, 0) mm, rotated rx -180 ry 0 rz -90 deg; joints [14.318, -114.153, -117.502, -38.345, 90, 14.318] of FAIRINO FR5
    - target Target_501 (Cartesian target) at (70, 30, 0) mm, rotated rx -180 ry 0 rz -90 deg; joints [14.595, -113.193, -119.135, -37.672, 90, 14.595] of FAIRINO FR5
    - target Target_502 (Cartesian target) at (60, 30, 0) mm, rotated rx -180 ry 0 rz -90 deg; joints [14.883, -112.232, -120.754, -37.014, 90, 14.883] of FAIRINO FR5
    - target Target_503 (Cartesian target) at (50, 30, 0) mm, rotated rx -180 ry 0 rz -90 deg; joints [15.183, -111.269, -122.361, -36.371, 90, 15.183] of FAIRINO FR5
    - target Target_504 (Cartesian target) at (40, 30, 0) mm, rotated rx -180 ry 0 rz -90 deg; joints [15.495, -110.302, -123.954, -35.744, 90, 15.495] of FAIRINO FR5
    - target Target_505 (Cartesian target) at (30, 30, 0) mm, rotated rx -180 ry 0 rz -90 deg; joints [15.821, -109.331, -125.537, -35.133, 90, 15.821] of FAIRINO FR5
    - target Target_506 (Cartesian target) at (20, 30, 0) mm, rotated rx -180 ry 0 rz -90 deg; joints [16.16, -108.354, -127.107, -34.539, 90, 16.16] of FAIRINO FR5
    - target Target_507 (Cartesian target) at (10, 30, 0) mm, rotated rx -180 ry 0 rz -90 deg; joints [16.515, -107.371, -128.667, -33.962, 90, 16.515] of FAIRINO FR5
    - target Target_508 (Cartesian target) at (0, 30, 0) mm, rotated rx -180 ry 0 rz -90 deg; joints [16.885, -106.38, -130.216, -33.404, 90, 16.885] of FAIRINO FR5
    - target Target_509 (Cartesian target) at (-10, 30, 0) mm, rotated rx -180 ry 0 rz -90 deg; joints [17.273, -105.379, -131.756, -32.865, 90, 17.273] of FAIRINO FR5
    - target Target_510 (Cartesian target) at (-20, 30, 0) mm, rotated rx -180 ry 0 rz -90 deg; joints [17.679, -104.368, -133.286, -32.347, 90, 17.679] of FAIRINO FR5
    - target Target_511 (Cartesian target) at (-30, 30, 0) mm, rotated rx -180 ry 0 rz -90 deg; joints [18.104, -103.344, -134.806, -31.85, 90, 18.104] of FAIRINO FR5
    - target Target_512 (Cartesian target) at (-40, 30, 0) mm, rotated rx -180 ry 0 rz -90 deg; joints [18.551, -102.306, -136.318, -31.377, 90, 18.551] of FAIRINO FR5
    - target Target_513 (Cartesian target) at (-50, 30, 0) mm, rotated rx -180 ry 0 rz -90 deg; joints [19.02, -101.251, -137.82, -30.929, 90, 19.02] of FAIRINO FR5
    - target Target_514 (Cartesian target) at (-60, 30, 0) mm, rotated rx -180 ry 0 rz -90 deg; joints [19.514, -100.177, -139.315, -30.509, 90, 19.514] of FAIRINO FR5
    - target Target_515 (Cartesian target) at (-70, 30, 0) mm, rotated rx -180 ry 0 rz -90 deg; joints [20.035, -99.081, -140.801, -30.118, 90, 20.035] of FAIRINO FR5
    - target Target_516 (Cartesian target) at (-80, 30, 0) mm, rotated rx -180 ry 0 rz -90 deg; joints [20.584, -97.961, -142.279, -29.76, 90, 20.584] of FAIRINO FR5
    - target Target_517 (Cartesian target) at (-90, 30, 0) mm, rotated rx -180 ry 0 rz -90 deg; joints [21.164, -96.812, -143.749, -29.438, 90, 21.164] of FAIRINO FR5
    - target Target_518 (Cartesian target) at (-100, 30, 0) mm, rotated rx -180 ry 0 rz -90 deg; joints [21.779, -95.631, -145.212, -29.157, 90, 21.779] of FAIRINO FR5
    - target Target_519 (Cartesian target) at (-110, 30, 0) mm, rotated rx -180 ry 0 rz -90 deg; joints [22.43, -94.413, -146.666, -28.921, 90, 22.43] of FAIRINO FR5
    - target Target_520 (Cartesian target) at (-120, 30, 0) mm, rotated rx -180 ry 0 rz -90 deg; joints [23.122, -93.152, -148.113, -28.735, 90, 23.122] of FAIRINO FR5
    - target Target_521 (Cartesian target) at (-130, 30, 0) mm, rotated rx -180 ry 0 rz -90 deg; joints [23.859, -91.842, -149.551, -28.607, 90, 23.859] of FAIRINO FR5
    - target Target_522 (Cartesian target) at (-140, 30, 0) mm, rotated rx -180 ry 0 rz -90 deg; joints [24.645, -90.475, -150.98, -28.545, 90, 24.645] of FAIRINO FR5
    - target Target_523 (Cartesian target) at (-140, 40, 0) mm, rotated rx -180 ry 0 rz -90 deg; joints [26.398, -90.632, -150.82, -28.548, 90, 26.398] of FAIRINO FR5
    - target Target_524 (Cartesian target) at (-130, 40, 0) mm, rotated rx -180 ry 0 rz -90 deg; joints [25.564, -91.988, -149.394, -28.618, 90, 25.564] of FAIRINO FR5
    - target Target_525 (Cartesian target) at (-120, 40, 0) mm, rotated rx -180 ry 0 rz -90 deg; joints [24.78, -93.288, -147.96, -28.752, 90, 24.78] of FAIRINO FR5
    - target Target_526 (Cartesian target) at (-110, 40, 0) mm, rotated rx -180 ry 0 rz -90 deg; joints [24.044, -94.54, -146.517, -28.943, 90, 24.044] of FAIRINO FR5
    - target Target_527 (Cartesian target) at (-100, 40, 0) mm, rotated rx -180 ry 0 rz -90 deg; joints [23.35, -95.751, -145.066, -29.183, 90, 23.35] of FAIRINO FR5
    - target Target_528 (Cartesian target) at (-90, 40, 0) mm, rotated rx -180 ry 0 rz -90 deg; joints [22.696, -96.925, -143.607, -29.468, 90, 22.696] of FAIRINO FR5
    - target Target_529 (Cartesian target) at (-80, 40, 0) mm, rotated rx -180 ry 0 rz -90 deg; joints [22.077, -98.068, -142.14, -29.792, 90, 22.077] of FAIRINO FR5
    - target Target_530 (Cartesian target) at (-70, 40, 0) mm, rotated rx -180 ry 0 rz -90 deg; joints [21.492, -99.183, -140.665, -30.152, 90, 21.492] of FAIRINO FR5
    - target Target_531 (Cartesian target) at (-60, 40, 0) mm, rotated rx -180 ry 0 rz -90 deg; joints [20.936, -100.274, -139.181, -30.545, 90, 20.936] of FAIRINO FR5
    - target Target_532 (Cartesian target) at (-50, 40, 0) mm, rotated rx -180 ry 0 rz -90 deg; joints [20.409, -101.344, -137.689, -30.967, 90, 20.409] of FAIRINO FR5
    - target Target_533 (Cartesian target) at (-40, 40, 0) mm, rotated rx -180 ry 0 rz -90 deg; joints [19.908, -102.395, -136.189, -31.416, 90, 19.908] of FAIRINO FR5
    - target Target_534 (Cartesian target) at (-30, 40, 0) mm, rotated rx -180 ry 0 rz -90 deg; joints [19.431, -103.43, -134.68, -31.89, 90, 19.431] of FAIRINO FR5
    - target Target_535 (Cartesian target) at (-20, 40, 0) mm, rotated rx -180 ry 0 rz -90 deg; joints [18.976, -104.451, -133.161, -32.388, 90, 18.976] of FAIRINO FR5
    - target Target_536 (Cartesian target) at (-10, 40, 0) mm, rotated rx -180 ry 0 rz -90 deg; joints [18.543, -105.459, -131.634, -32.907, 90, 18.543] of FAIRINO FR5
    - target Target_537 (Cartesian target) at (0, 40, 0) mm, rotated rx -180 ry 0 rz -90 deg; joints [18.128, -106.457, -130.096, -33.446, 90, 18.128] of FAIRINO FR5
    - target Target_538 (Cartesian target) at (10, 40, 0) mm, rotated rx -180 ry 0 rz -90 deg; joints [17.732, -107.446, -128.549, -34.005, 90, 17.732] of FAIRINO FR5
    - target Target_539 (Cartesian target) at (20, 40, 0) mm, rotated rx -180 ry 0 rz -90 deg; joints [17.353, -108.427, -126.991, -34.582, 90, 17.353] of FAIRINO FR5
    - target Target_540 (Cartesian target) at (30, 40, 0) mm, rotated rx -180 ry 0 rz -90 deg; joints [16.99, -109.402, -125.422, -35.177, 90, 16.99] of FAIRINO FR5
    - target Target_541 (Cartesian target) at (40, 40, 0) mm, rotated rx -180 ry 0 rz -90 deg; joints [16.641, -110.371, -123.841, -35.788, 90, 16.641] of FAIRINO FR5
    - target Target_542 (Cartesian target) at (50, 40, 0) mm, rotated rx -180 ry 0 rz -90 deg; joints [16.307, -111.336, -122.249, -36.415, 90, 16.307] of FAIRINO FR5
    - target Target_543 (Cartesian target) at (60, 40, 0) mm, rotated rx -180 ry 0 rz -90 deg; joints [15.986, -112.298, -120.644, -37.058, 90, 15.986] of FAIRINO FR5
    - target Target_544 (Cartesian target) at (70, 40, 0) mm, rotated rx -180 ry 0 rz -90 deg; joints [15.677, -113.258, -119.025, -37.717, 90, 15.677] of FAIRINO FR5
    - target Target_545 (Cartesian target) at (80, 40, 0) mm, rotated rx -180 ry 0 rz -90 deg; joints [15.38, -114.216, -117.393, -38.39, 90, 15.38] of FAIRINO FR5
    - target Target_546 (Cartesian target) at (90, 40, 0) mm, rotated rx -180 ry 0 rz -90 deg; joints [15.094, -115.174, -115.747, -39.078, 90, 15.094] of FAIRINO FR5
    - target Target_547 (Cartesian target) at (100, 40, 0) mm, rotated rx -180 ry 0 rz -90 deg; joints [14.819, -116.133, -114.086, -39.781, 90, 14.819] of FAIRINO FR5
    - target Target_548 (Cartesian target) at (110, 40, 0) mm, rotated rx -180 ry 0 rz -90 deg; joints [14.553, -117.093, -112.409, -40.499, 90, 14.553] of FAIRINO FR5
    - target Target_549 (Cartesian target) at (120, 40, 0) mm, rotated rx -180 ry 0 rz -90 deg; joints [14.297, -118.054, -110.715, -41.231, 90, 14.297] of FAIRINO FR5
    - target Target_550 (Cartesian target) at (130, 40, 0) mm, rotated rx -180 ry 0 rz -90 deg; joints [14.05, -119.019, -109.003, -41.978, 90, 14.05] of FAIRINO FR5
    - target Target_551 (Cartesian target) at (140, 40, 0) mm, rotated rx -180 ry 0 rz -90 deg; joints [13.811, -119.987, -107.273, -42.739, 90, 13.811] of FAIRINO FR5
    - target Target_552 (Cartesian target) at (140, 50, 0) mm, rotated rx -180 ry 0 rz -90 deg; joints [14.763, -120.061, -107.141, -42.798, 90, 14.763] of FAIRINO FR5
    - target Target_553 (Cartesian target) at (130, 50, 0) mm, rotated rx -180 ry 0 rz -90 deg; joints [15.018, -119.094, -108.87, -42.036, 90, 15.018] of FAIRINO FR5
    - target Target_554 (Cartesian target) at (120, 50, 0) mm, rotated rx -180 ry 0 rz -90 deg; joints [15.282, -118.13, -110.58, -41.289, 90, 15.282] of FAIRINO FR5
    - target Target_555 (Cartesian target) at (110, 50, 0) mm, rotated rx -180 ry 0 rz -90 deg; joints [15.555, -117.17, -112.273, -40.557, 90, 15.555] of FAIRINO FR5
    - target Target_556 (Cartesian target) at (100, 50, 0) mm, rotated rx -180 ry 0 rz -90 deg; joints [15.838, -116.211, -113.949, -39.839, 90, 15.838] of FAIRINO FR5
    - target Target_557 (Cartesian target) at (90, 50, 0) mm, rotated rx -180 ry 0 rz -90 deg; joints [16.131, -115.254, -115.609, -39.136, 90, 16.131] of FAIRINO FR5
    - target Target_558 (Cartesian target) at (80, 50, 0) mm, rotated rx -180 ry 0 rz -90 deg; joints [16.436, -114.298, -117.254, -38.448, 90, 16.436] of FAIRINO FR5
    - target Target_559 (Cartesian target) at (70, 50, 0) mm, rotated rx -180 ry 0 rz -90 deg; joints [16.752, -113.341, -118.885, -37.774, 90, 16.752] of FAIRINO FR5
    - target Target_560 (Cartesian target) at (60, 50, 0) mm, rotated rx -180 ry 0 rz -90 deg; joints [17.08, -112.383, -120.501, -37.116, 90, 17.08] of FAIRINO FR5
    - target Target_561 (Cartesian target) at (50, 50, 0) mm, rotated rx -180 ry 0 rz -90 deg; joints [17.422, -111.423, -122.105, -36.472, 90, 17.422] of FAIRINO FR5
    - target Target_562 (Cartesian target) at (40, 50, 0) mm, rotated rx -180 ry 0 rz -90 deg; joints [17.778, -110.46, -123.695, -35.845, 90, 17.778] of FAIRINO FR5
    - target Target_563 (Cartesian target) at (30, 50, 0) mm, rotated rx -180 ry 0 rz -90 deg; joints [18.149, -109.493, -125.274, -35.233, 90, 18.149] of FAIRINO FR5
    - target Target_564 (Cartesian target) at (20, 50, 0) mm, rotated rx -180 ry 0 rz -90 deg; joints [18.535, -108.521, -126.841, -34.638, 90, 18.535] of FAIRINO FR5
    - target Target_565 (Cartesian target) at (10, 50, 0) mm, rotated rx -180 ry 0 rz -90 deg; joints [18.938, -107.542, -128.397, -34.061, 90, 18.938] of FAIRINO FR5
    - target Target_566 (Cartesian target) at (0, 50, 0) mm, rotated rx -180 ry 0 rz -90 deg; joints [19.36, -106.556, -129.942, -33.501, 90, 19.36] of FAIRINO FR5
    - target Target_567 (Cartesian target) at (-10, 50, 0) mm, rotated rx -180 ry 0 rz -90 deg; joints [19.8, -105.562, -131.477, -32.961, 90, 19.8] of FAIRINO FR5
    - target Target_568 (Cartesian target) at (-20, 50, 0) mm, rotated rx -180 ry 0 rz -90 deg; joints [20.261, -104.557, -133.002, -32.441, 90, 20.261] of FAIRINO FR5
    - target Target_569 (Cartesian target) at (-30, 50, 0) mm, rotated rx -180 ry 0 rz -90 deg; joints [20.744, -103.54, -134.518, -31.943, 90, 20.744] of FAIRINO FR5
    - target Target_570 (Cartesian target) at (-40, 50, 0) mm, rotated rx -180 ry 0 rz -90 deg; joints [21.25, -102.509, -136.024, -31.467, 90, 21.25] of FAIRINO FR5
    - target Target_571 (Cartesian target) at (-50, 50, 0) mm, rotated rx -180 ry 0 rz -90 deg; joints [21.782, -101.463, -137.521, -31.016, 90, 21.782] of FAIRINO FR5
    - target Target_572 (Cartesian target) at (-60, 50, 0) mm, rotated rx -180 ry 0 rz -90 deg; joints [22.341, -100.398, -139.01, -30.592, 90, 22.341] of FAIRINO FR5
    - target Target_573 (Cartesian target) at (-70, 50, 0) mm, rotated rx -180 ry 0 rz -90 deg; joints [22.93, -99.313, -140.49, -30.197, 90, 22.93] of FAIRINO FR5
    - target Target_574 (Cartesian target) at (-80, 50, 0) mm, rotated rx -180 ry 0 rz -90 deg; joints [23.55, -98.205, -141.961, -29.834, 90, 23.55] of FAIRINO FR5
    - target Target_575 (Cartesian target) at (-90, 50, 0) mm, rotated rx -180 ry 0 rz -90 deg; joints [24.206, -97.069, -143.424, -29.506, 90, 24.206] of FAIRINO FR5
    - target Target_576 (Cartesian target) at (-100, 50, 0) mm, rotated rx -180 ry 0 rz -90 deg; joints [24.898, -95.903, -144.879, -29.217, 90, 24.898] of FAIRINO FR5
    - target Target_577 (Cartesian target) at (-110, 50, 0) mm, rotated rx -180 ry 0 rz -90 deg; joints [25.632, -94.702, -146.326, -28.972, 90, 25.632] of FAIRINO FR5
    - target Target_578 (Cartesian target) at (-120, 50, 0) mm, rotated rx -180 ry 0 rz -90 deg; joints [26.41, -93.461, -147.764, -28.775, 90, 26.41] of FAIRINO FR5
    - target Target_579 (Cartesian target) at (-130, 50, 0) mm, rotated rx -180 ry 0 rz -90 deg; joints [27.237, -92.174, -149.193, -28.633, 90, 27.237] of FAIRINO FR5
    - target Target_580 (Cartesian target) at (-140, 50, 0) mm, rotated rx -180 ry 0 rz -90 deg; joints [28.118, -90.832, -150.614, -28.554, 90, 28.118] of FAIRINO FR5
    - target Target_581 (Cartesian target) at (-140, 60, 0) mm, rotated rx -180 ry 0 rz -90 deg; joints [29.801, -91.074, -150.363, -28.563, 90, 29.801] of FAIRINO FR5
    - target Target_582 (Cartesian target) at (-130, 60, 0) mm, rotated rx -180 ry 0 rz -90 deg; joints [28.877, -92.398, -148.949, -28.653, 90, 28.877] of FAIRINO FR5
    - target Target_583 (Cartesian target) at (-120, 60, 0) mm, rotated rx -180 ry 0 rz -90 deg; joints [28.009, -93.671, -147.526, -28.804, 90, 28.009] of FAIRINO FR5
    - target Target_584 (Cartesian target) at (-110, 60, 0) mm, rotated rx -180 ry 0 rz -90 deg; joints [27.192, -94.899, -146.093, -29.008, 90, 27.192] of FAIRINO FR5
    - target Target_585 (Cartesian target) at (-100, 60, 0) mm, rotated rx -180 ry 0 rz -90 deg; joints [26.42, -96.088, -144.652, -29.26, 90, 26.42] of FAIRINO FR5
    - target Target_586 (Cartesian target) at (-90, 60, 0) mm, rotated rx -180 ry 0 rz -90 deg; joints [25.691, -97.244, -143.202, -29.554, 90, 25.691] of FAIRINO FR5
    - target Target_587 (Cartesian target) at (-80, 60, 0) mm, rotated rx -180 ry 0 rz -90 deg; joints [25.002, -98.371, -141.743, -29.886, 90, 25.002] of FAIRINO FR5
    - target Target_588 (Cartesian target) at (-70, 60, 0) mm, rotated rx -180 ry 0 rz -90 deg; joints [24.348, -99.471, -140.276, -30.252, 90, 24.348] of FAIRINO FR5
    - target Target_589 (Cartesian target) at (-60, 60, 0) mm, rotated rx -180 ry 0 rz -90 deg; joints [23.727, -100.549, -138.801, -30.65, 90, 23.727] of FAIRINO FR5
    - target Target_590 (Cartesian target) at (-50, 60, 0) mm, rotated rx -180 ry 0 rz -90 deg; joints [23.137, -101.607, -137.316, -31.077, 90, 23.137] of FAIRINO FR5
    - target Target_591 (Cartesian target) at (-40, 60, 0) mm, rotated rx -180 ry 0 rz -90 deg; joints [22.576, -102.648, -135.823, -31.529, 90, 22.576] of FAIRINO FR5
    - target Target_592 (Cartesian target) at (-30, 60, 0) mm, rotated rx -180 ry 0 rz -90 deg; joints [22.041, -103.673, -134.32, -32.007, 90, 22.041] of FAIRINO FR5
